gfCNCPoint4[1229] = {X 18.0872, Y 34.0798, Z -5.5000, A 0.000, B 0.000, C 0.000 }
gfCNCPoint4[1230] = {X 16.0874, Y 34.3007, Z -5.5000, A 0.000, B 0.000, C 0.000 }
gfCNCPoint4[1231] = {X 15.3633, Y 34.3534, Z -5.5000, A 0.000, B 0.000, C 0.000 }
gfCNCPoint4[1232] = {X 14.6390, Y 34.4040, Z -5.5000, A 0.000, B 0.000, C 0.000 }
gfCNCPoint4[1233] = {X 10.6873, Y 35.0236, Z -5.5000, A 0.000, B 0.000, C 0.000 }
gfCNCPoint4[1234] = {X 14.7700, Y 36.3195, Z -5.5000, A 0.000, B 0.000, C 0.000 }
gfCNCPoint4[1235] = {X 14.6336, Y 34.3242, Z -5.5000, A 0.000, B 0.000, C 0.000 }
gfCNCPoint4[1236] = {X 12.2421, Y 34.4763, Z -5.5000, A 0.000, B 0.000, C 0.000 }
gfCNCPoint4[1237] = {X 9.8492, Y 34.6056, Z -5.5000, A 0.000, B 0.000, C 0.000 }
gfCNCPoint4[1238] = {X 8.5938, Y 34.7145, Z -5.5000, A 0.000, B 0.000, C 0.000 }
gfCNCPoint4[1239] = {X 7.3613, Y 34.9767, Z -5.5000, A 0.000, B 0.000, C 0.000 }
gfCNCPoint4[1240] = {X 7.2805, Y 35.1981, Z -5.5000, A 0.000, B 0.000, C 0.000 }
gfCNCPoint4[1241] = {X 7.2526, Y 35.4321, Z -5.5000, A 0.000, B 0.000, C 0.000 }
gfCNCPoint4[1242] = {X 7.3219, Y 35.9823, Z -5.5000, A 0.000, B 0.000, C 0.000 }
gfCNCPoint4[1243] = {X 7.5291, Y 36.4967, Z -5.5000, A 0.000, B 0.000, C 0.000 }
gfCNCPoint4[1244] = {X 7.8606, Y 36.9413, Z -5.5000, A 0.000, B 0.000, C 0.000 }
gfCNCPoint4[1245] = {X 8.2944, Y 37.2868, Z -5.5000, A 0.000, B 0.000, C 0.000 }
gfCNCPoint4[1246] = {X 9.1221, Y 37.7063, Z -5.5000, A 0.000, B 0.000, C 0.000 }
gfCNCPoint4[1247] = {X 10.0031, Y 37.9977, Z -5.5000, A 0.000, B 0.000, C 0.000 }
gfCNCPoint4[1248] = {X 11.3365, Y 38.2429, Z -5.5000, A 0.000, B 0.000, C 0.000 }
gfCNCPoint4[1249] = {X 12.6902, Y 38.3190, Z -5.5000, A 0.000, B 0.000, C 0.000 }
gfCNCPoint4[1250] = {X 14.0427, Y 38.2248, Z -5.5000, A 0.000, B 0.000, C 0.000 }
gfCNCPoint4[1251] = {X 15.3727, Y 37.9617, Z -5.5000, A 0.000, B 0.000, C 0.000 }
gfCNCPoint4[1252] = {X 16.6593, Y 37.5340, Z -5.5000, A 0.000, B 0.000, C 0.000 }
gfCNCPoint4[1253] = {X 18.0880, Y 36.8591, Z -5.5000, A 0.000, B 0.000, C 0.000 }
gfCNCPoint4[1254] = {X 19.4300, Y 36.0248, Z -5.5000, A 0.000, B 0.000, C 0.000 }
gfCNCPoint4[1255] = {X 19.5226, Y 35.1553, Z -5.5000, A 0.000, B 0.000, C 0.000 }
gfCNCPoint4[1256] = {X 19.8019, Y 34.3266, Z -5.5000, A 0.000, B 0.000, C 0.000 }
gfCNCPoint4[1257] = {X 20.2547, Y 33.5784, Z -5.5000, A 0.000, B 0.000, C 0.000 }
gfCNCPoint4[1258] = {X 18.1812, Y 33.9846, Z -5.5000, A 0.000, B 0.000, C 0.000 }
gfCNCPoint4[1259] = {X 16.0816, Y 34.2210, Z -5.5000, A 0.000, B 0.000, C 0.000 }
gfCNCPoint4[1260] = {X 15.3577, Y 34.2736, Z -5.5000, A 0.000, B 0.000, C 0.000 }
gfCNCPoint4[1261] = {X 14.6336, Y 34.3242, Z -5.5000, A 0.000, B 0.000, C 0.000 }
gfCNCPoint4[1262] = {X 14.7700, Y 36.3195, Z -5.5000, A 0.000, B 0.000, C 0.000 }
gfCNCPoint4[1263] = {X 14.7700, Y 36.3195, Z -2.5000, A 0.000, B 0.000, C 0.000 }
gfCNCPoint4[1264] = {X 14.7700, Y 36.3195, Z 11.0000, A 0.000, B 0.000, C 0.000 }
gfCNCPoint4[1265] = {X 165.6772, Y 73.8165, Z 11.0000, A 0.000, B 0.000, C 0.000 }
gfCNCPoint4[1266] = {X 165.6772, Y 73.8165, Z -1.6667, A 0.000, B 0.000, C 0.000 }
gfCNCPoint4[1267] = {X 161.3996, Y 78.5670, Z -3.3796, A 0.000, B 0.000, C 0.000 }
gfCNCPoint4[1268] = {X 169.3132, Y 78.5670, Z -5.5000, A 0.000, B 0.000, C 0.000 }
gfCNCPoint4[1269] = {X 169.3132, Y 76.1670, Z -5.5000, A 0.000, B 0.000, C 0.000 }
gfCNCPoint4[1270] = {X 171.8361, Y 76.1670, Z -5.5000, A 0.000, B 0.000, C 0.000 }
gfCNCPoint4[1271] = {X 169.3147, Y 73.3634, Z -5.5000, A 0.000, B 0.000, C 0.000 }
gfCNCPoint4[1272] = {X 166.7903, Y 76.1670, Z -5.5000, A 0.000, B 0.000, C 0.000 }
gfCNCPoint4[1273] = {X 169.3132, Y 76.1670, Z -5.5000, A 0.000, B 0.000, C 0.000 }
gfCNCPoint4[1274] = {X 169.3132, Y 78.5670, Z -5.5000, A 0.000, B 0.000, C 0.000 }
gfCNCPoint4[1275] = {X 177.2224, Y 78.5670, Z -5.5000, A 0.000, B 0.000, C 0.000 }
gfCNCPoint4[1276] = {X 169.3158, Y 69.7756, Z -5.5000, A 0.000, B 0.000, C 0.000 }
gfCNCPoint4[1277] = {X 161.3996, Y 78.5670, Z -5.5000, A 0.000, B 0.000, C 0.000 }
gfCNCPoint4[1278] = {X 169.3132, Y 78.5670, Z -5.5000, A 0.000, B 0.000, C 0.000 }
gfCNCPoint4[1279] = {X 169.3132, Y 74.6470, Z -5.5000, A 0.000, B 0.000, C 0.000 }
gfCNCPoint4[1280] = {X 169.3132, Y 78.6470, Z -5.5000, A 0.000, B 0.000, C 0.000 }
gfCNCPoint4[1281] = {X 177.4019, Y 78.6470, Z -5.5000, A 0.000, B 0.000, C 0.000 }
gfCNCPoint4[1282] = {X 169.3159, Y 69.6560, Z -5.5000, A 0.000, B 0.000, C 0.000 }
gfCNCPoint4[1283] = {X 161.2199, Y 78.6470, Z -5.5000, A 0.000, B 0.000, C 0.000 }
gfCNCPoint4[1284] = {X 169.3132, Y 78.6470, Z -5.5000, A 0.000, B 0.000, C 0.000 }
gfCNCPoint4[1285] = {X 169.3132, Y 74.6470, Z -5.5000, A 0.000, B 0.000, C 0.000 }
gfCNCPoint4[1286] = {X 169.3132, Y 74.7270, Z -5.5000, A 0.000, B 0.000, C 0.000 }
gfCNCPoint4[1287] = {X 169.3132, Y 78.7270, Z -5.5000, A 0.000, B 0.000, C 0.000 }
gfCNCPoint4[1288] = {X 177.5814, Y 78.7270, Z -5.5000, A 0.000, B 0.000, C 0.000 }
gfCNCPoint4[1289] = {X 169.3159, Y 69.5364, Z -5.5000, A 0.000, B 0.000, C 0.000 }
gfCNCPoint4[1290] = {X 161.0403, Y 78.7270, Z -5.5000, A 0.000, B 0.000, C 0.000 }
gfCNCPoint4[1291] = {X 169.3132, Y 78.7270, Z -5.5000, A 0.000, B 0.000, C 0.000 }
gfCNCPoint4[1292] = {X 169.3132, Y 74.7270, Z -5.5000, A 0.000, B 0.000, C 0.000 }
gfCNCPoint4[1293] = {X 169.3132, Y 74.8070, Z -5.5000, A 0.000, B 0.000, C 0.000 }
gfCNCPoint4[1294] = {X 169.3132, Y 78.8070, Z -5.5000, A 0.000, B 0.000, C 0.000 }
gfCNCPoint4[1295] = {X 177.7610, Y 78.8070, Z -5.5000, A 0.000, B 0.000, C 0.000 }
gfCNCPoint4[1296] = {X 169.3159, Y 69.4168, Z -5.5000, A 0.000, B 0.000, C 0.000 }
gfCNCPoint4[1297] = {X 160.8606, Y 78.8070, Z -5.5000, A 0.000, B 0.000, C 0.000 }
gfCNCPoint4[1298] = {X 169.3132, Y 78.8070, Z -5.5000, A 0.000, B 0.000, C 0.000 }
gfCNCPoint4[1299] = {X 169.3132, Y 74.8070, Z -5.5000, A 0.000, B 0.000, C 0.000 }
gfCNCPoint4[1300] = {X 169.3132, Y 74.8870, Z -5.5000, A 0.000, B 0.000, C 0.000 }
gfCNCPoint4[1301] = {X 169.3132, Y 78.8870, Z -5.5000, A 0.000, B 0.000, C 0.000 }
gfCNCPoint4[1302] = {X 177.9405, Y 78.8870, Z -5.5000, A 0.000, B 0.000, C 0.000 }
gfCNCPoint4[1303] = {X 169.3160, Y 69.2972, Z -5.5000, A 0.000, B 0.000, C 0.000 }
gfCNCPoint4[1304] = {X 160.6809, Y 78.8870, Z -5.5000, A 0.000, B 0.000, C 0.000 }
gfCNCPoint4[1305] = {X 169.3132, Y 78.8870, Z -5.5000, A 0.000, B 0.000, C 0.000 }
gfCNCPoint4[1306] = {X 169.3132, Y 74.8870, Z -5.5000, A 0.000, B 0.000, C 0.000 }
gfCNCPoint4[1307] = {X 169.3132, Y 74.9670, Z -5.5000, A 0.000, B 0.000, C 0.000 }
gfCNCPoint4[1308] = {X 169.3132, Y 78.9670, Z -5.5000, A 0.000, B 0.000, C 0.000 }
gfCNCPoint4[1309] = {X 178.1201, Y 78.9670, Z -5.5000, A 0.000, B 0.000, C 0.000 }
gfCNCPoint4[1310] = {X 169.3160, Y 69.1776, Z -5.5000, A 0.000, B 0.000, C 0.000 }
gfCNCPoint4[1311] = {X 160.5012, Y 78.9670, Z -5.5000, A 0.000, B 0.000, C 0.000 }
gfCNCPoint4[1312] = {X 169.3132, Y 78.9670, Z -5.5000, A 0.000, B 0.000, C 0.000 }
gfCNCPoint4[1313] = {X 169.3132, Y 74.9670, Z -5.5000, A 0.000, B 0.000, C 0.000 }
gfCNCPoint4[1314] = {X 169.3132, Y 74.9670, Z -2.5000, A 0.000, B 0.000, C 0.000 }
gfCNCPoint4[1315] = {X 169.3132, Y 74.9670, Z 11.0000, A 0.000, B 0.000, C 0.000 }
gfCNCPoint4[1316] = {X 186.2281, Y 37.9121, Z 11.0000, A 0.000, B 0.000, C 0.000 }
gfCNCPoint4[1317] = {X 186.2281, Y 37.9121, Z -1.6667, A 0.000, B 0.000, C 0.000 }
gfCNCPoint4[1318] = {X 187.5897, Y 37.8323, Z -2.0321, A 0.000, B 0.000, C 0.000 }
gfCNCPoint4[1319] = {X 189.4169, Y 37.3859, Z -2.5361, A 0.000, B 0.000, C 0.000 }
gfCNCPoint4[1320] = {X 190.1421, Y 37.0740, Z -2.7476, A 0.000, B 0.000, C 0.000 }
gfCNCPoint4[1321] = {X 190.9803, Y 36.7135, Z -2.9922, A 0.000, B 0.000, C 0.000 }
gfCNCPoint4[1322] = {X 191.6914, Y 36.3240, Z -3.2094, A 0.000, B 0.000, C 0.000 }
gfCNCPoint4[1323] = {X 192.4466, Y 35.8118, Z -3.4539, A 0.000, B 0.000, C 0.000 }
gfCNCPoint4[1324] = {X 192.4699, Y 35.2976, Z -3.5918, A 0.000, B 0.000, C 0.000 }
gfCNCPoint4[1325] = {X 192.6312, Y 34.6351, Z -3.7745, A 0.000, B 0.000, C 0.000 }
gfCNCPoint4[1326] = {X 192.8468, Y 34.1677, Z -3.9124, A 0.000, B 0.000, C 0.000 }
gfCNCPoint4[1327] = {X 192.7389, Y 34.1929, Z -3.9421, A 0.000, B 0.000, C 0.000 }
gfCNCPoint4[1328] = {X 191.4080, Y 34.4432, Z -4.3050, A 0.000, B 0.000, C 0.000 }
gfCNCPoint4[1329] = {X 190.5815, Y 34.5495, Z -4.5283, A 0.000, B 0.000, C 0.000 }
gfCNCPoint4[1330] = {X 189.2271, Y 34.6445, Z -4.8921, A 0.000, B 0.000, C 0.000 }
gfCNCPoint4[1331] = {X 186.9627, Y 34.7836, Z -5.5000, A 0.000, B 0.000, C 0.000 }
gfCNCPoint4[1332] = {X 182.5757, Y 35.0529, Z -5.5000, A 0.000, B 0.000, C 0.000 }
gfCNCPoint4[1333] = {X 181.8176, Y 35.1403, Z -5.5000, A 0.000, B 0.000, C 0.000 }
gfCNCPoint4[1334] = {X 181.0731, Y 35.3082, Z -5.5000, A 0.000, B 0.000, C 0.000 }
gfCNCPoint4[1335] = {X 181.0650, Y 35.3823, Z -5.5000, A 0.000, B 0.000, C 0.000 }
gfCNCPoint4[1336] = {X 181.0651, Y 35.4570, Z -5.5000, A 0.000, B 0.000, C 0.000 }
gfCNCPoint4[1337] = {X 181.1578, Y 35.9998, Z -5.5000, A 0.000, B 0.000, C 0.000 }
gfCNCPoint4[1338] = {X 181.4149, Y 36.4869, Z -5.5000, A 0.000, B 0.000, C 0.000 }
gfCNCPoint4[1339] = {X 181.8107, Y 36.8698, Z -5.5000, A 0.000, B 0.000, C 0.000 }
gfCNCPoint4[1340] = {X 182.4284, Y 37.2226, Z -5.5000, A 0.000, B 0.000, C 0.000 }
gfCNCPoint4[1341] = {X 183.0886, Y 37.4872, Z -5.5000, A 0.000, B 0.000, C 0.000 }
gfCNCPoint4[1342] = {X 184.4948, Y 37.8011, Z -5.5000, A 0.000, B 0.000, C 0.000 }
gfCNCPoint4[1343] = {X 185.9310, Y 37.9170, Z -5.5000, A 0.000, B 0.000, C 0.000 }
gfCNCPoint4[1344] = {X 187.3693, Y 37.8327, Z -5.5000, A 0.000, B 0.000, C 0.000 }
gfCNCPoint4[1345] = {X 188.7821, Y 37.5499, Z -5.5000, A 0.000, B 0.000, C 0.000 }
gfCNCPoint4[1346] = {X 190.1421, Y 37.0740, Z -5.5000, A 0.000, B 0.000, C 0.000 }
gfCNCPoint4[1347] = {X 191.3243, Y 36.4976, Z -5.5000, A 0.000, B 0.000, C 0.000 }
gfCNCPoint4[1348] = {X 192.4466, Y 35.8118, Z -5.5000, A 0.000, B 0.000, C 0.000 }
gfCNCPoint4[1349] = {X 192.5670, Y 34.9703, Z -5.5000, A 0.000, B 0.000, C 0.000 }
gfCNCPoint4[1350] = {X 192.8468, Y 34.1677, Z -5.5000, A 0.000, B 0.000, C 0.000 }
gfCNCPoint4[1351] = {X 192.7389, Y 34.1929, Z -5.5000, A 0.000, B 0.000, C 0.000 }
gfCNCPoint4[1352] = {X 190.9895, Y 34.4696, Z -5.5000, A 0.000, B 0.000, C 0.000 }
gfCNCPoint4[1353] = {X 189.2271, Y 34.6445, Z -5.5000, A 0.000, B 0.000, C 0.000 }
gfCNCPoint4[1354] = {X 186.9627, Y 34.7836, Z -5.5000, A 0.000, B 0.000, C 0.000 }
gfCNCPoint4[1355] = {X 190.9564, Y 34.8075, Z -5.5000, A 0.000, B 0.000, C 0.000 }
gfCNCPoint4[1356] = {X 186.9578, Y 34.7037, Z -5.5000, A 0.000, B 0.000, C 0.000 }
gfCNCPoint4[1357] = {X 182.5708, Y 34.9731, Z -5.5000, A 0.000, B 0.000, C 0.000 }
gfCNCPoint4[1358] = {X 181.7800, Y 35.0656, Z -5.5000, A 0.000, B 0.000, C 0.000 }
gfCNCPoint4[1359] = {X 181.0042, Y 35.2447, Z -5.5000, A 0.000, B 0.000, C 0.000 }
gfCNCPoint4[1360] = {X 180.9874, Y 35.3482, Z -5.5000, A 0.000, B 0.000, C 0.000 }
gfCNCPoint4[1361] = {X 180.9850, Y 35.4530, Z -5.5000, A 0.000, B 0.000, C 0.000 }
gfCNCPoint4[1362] = {X 181.0811, Y 36.0228, Z -5.5000, A 0.000, B 0.000, C 0.000 }
gfCNCPoint4[1363] = {X 181.3503, Y 36.5341, Z -5.5000, A 0.000, B 0.000, C 0.000 }
gfCNCPoint4[1364] = {X 181.7656, Y 36.9358, Z -5.5000, A 0.000, B 0.000, C 0.000 }
gfCNCPoint4[1365] = {X 182.3936, Y 37.2947, Z -5.5000, A 0.000, B 0.000, C 0.000 }
gfCNCPoint4[1366] = {X 183.0649, Y 37.5636, Z -5.5000, A 0.000, B 0.000, C 0.000 }
gfCNCPoint4[1367] = {X 184.4822, Y 37.8801, Z -5.5000, A 0.000, B 0.000, C 0.000 }
gfCNCPoint4[1368] = {X 185.9296, Y 37.9970, Z -5.5000, A 0.000, B 0.000, C 0.000 }
gfCNCPoint4[1369] = {X 187.3792, Y 37.9121, Z -5.5000, A 0.000, B 0.000, C 0.000 }
gfCNCPoint4[1370] = {X 188.8031, Y 37.6271, Z -5.5000, A 0.000, B 0.000, C 0.000 }
gfCNCPoint4[1371] = {X 190.1737, Y 37.1475, Z -5.5000, A 0.000, B 0.000, C 0.000 }
gfCNCPoint4[1372] = {X 191.3805, Y 36.5581, Z -5.5000, A 0.000, B 0.000, C 0.000 }
gfCNCPoint4[1373] = {X 192.5249, Y 35.8553, Z -5.5000, A 0.000, B 0.000, C 0.000 }
gfCNCPoint4[1374] = {X 192.6602, Y 34.9276, Z -5.5000, A 0.000, B 0.000, C 0.000 }
gfCNCPoint4[1375] = {X 192.9924, Y 34.0510, Z -5.5000, A 0.000, B 0.000, C 0.000 }
gfCNCPoint4[1376] = {X 192.7315, Y 34.1128, Z -5.5000, A 0.000, B 0.000, C 0.000 }
gfCNCPoint4[1377] = {X 190.9841, Y 34.3897, Z -5.5000, A 0.000, B 0.000, C 0.000 }
gfCNCPoint4[1378] = {X 189.2236, Y 34.5646, Z -5.5000, A 0.000, B 0.000, C 0.000 }
gfCNCPoint4[1379] = {X 186.9578, Y 34.7037, Z -5.5000, A 0.000, B 0.000, C 0.000 }
gfCNCPoint4[1380] = {X 183.0018, Y 35.2959, Z -5.5000, A 0.000, B 0.000, C 0.000 }
gfCNCPoint4[1381] = {X 190.9515, Y 34.7276, Z -5.5000, A 0.000, B 0.000, C 0.000 }
gfCNCPoint4[1382] = {X 186.9529, Y 34.6239, Z -5.5000, A 0.000, B 0.000, C 0.000 }
gfCNCPoint4[1383] = {X 182.5658, Y 34.8932, Z -5.5000, A 0.000, B 0.000, C 0.000 }
gfCNCPoint4[1384] = {X 181.7439, Y 34.9907, Z -5.5000, A 0.000, B 0.000, C 0.000 }
gfCNCPoint4[1385] = {X 180.9383, Y 35.1806, Z -5.5000, A 0.000, B 0.000, C 0.000 }
gfCNCPoint4[1386] = {X 180.9104, Y 35.3165, Z -5.5000, A 0.000, B 0.000, C 0.000 }
gfCNCPoint4[1387] = {X 180.9051, Y 35.4551, Z -5.5000, A 0.000, B 0.000, C 0.000 }
gfCNCPoint4[1388] = {X 181.0057, Y 36.0496, Z -5.5000, A 0.000, B 0.000, C 0.000 }
gfCNCPoint4[1389] = {X 181.2869, Y 36.5829, Z -5.5000, A 0.000, B 0.000, C 0.000 }
gfCNCPoint4[1390] = {X 181.7205, Y 37.0019, Z -5.5000, A 0.000, B 0.000, C 0.000 }
gfCNCPoint4[1391] = {X 182.3588, Y 37.3667, Z -5.5000, A 0.000, B 0.000, C 0.000 }
gfCNCPoint4[1392] = {X 183.0413, Y 37.6400, Z -5.5000, A 0.000, B 0.000, C 0.000 }
gfCNCPoint4[1393] = {X 184.4695, Y 37.9591, Z -5.5000, A 0.000, B 0.000, C 0.000 }
gfCNCPoint4[1394] = {X 185.9281, Y 38.0770, Z -5.5000, A 0.000, B 0.000, C 0.000 }
gfCNCPoint4[1395] = {X 187.3890, Y 37.9915, Z -5.5000, A 0.000, B 0.000, C 0.000 }
gfCNCPoint4[1396] = {X 188.8240, Y 37.7043, Z -5.5000, A 0.000, B 0.000, C 0.000 }
gfCNCPoint4[1397] = {X 190.2053, Y 37.2210, Z -5.5000, A 0.000, B 0.000, C 0.000 }
gfCNCPoint4[1398] = {X 191.4368, Y 36.6184, Z -5.5000, A 0.000, B 0.000, C 0.000 }
gfCNCPoint4[1399] = {X 192.6036, Y 35.8984, Z -5.5000, A 0.000, B 0.000, C 0.000 }
gfCNCPoint4[1400] = {X 192.6773, Y 35.2164, Z -5.5000, A 0.000, B 0.000, C 0.000 }
gfCNCPoint4[1401] = {X 192.8599, Y 34.5552, Z -5.5000, A 0.000, B 0.000, C 0.000 }
gfCNCPoint4[1402] = {X 193.1467, Y 33.9322, Z -5.5000, A 0.000, B 0.000, C 0.000 }
gfCNCPoint4[1403] = {X 192.7149, Y 34.0346, Z -5.5000, A 0.000, B 0.000, C 0.000 }
gfCNCPoint4[1404] = {X 190.9731, Y 34.3104, Z -5.5000, A 0.000, B 0.000, C 0.000 }
gfCNCPoint4[1405] = {X 189.2183, Y 34.4848, Z -5.5000, A 0.000, B 0.000, C 0.000 }
gfCNCPoint4[1406] = {X 186.9529, Y 34.6239, Z -5.5000, A 0.000, B 0.000, C 0.000 }
gfCNCPoint4[1407] = {X 182.9969, Y 35.2160, Z -5.5000, A 0.000, B 0.000, C 0.000 }
gfCNCPoint4[1408] = {X 190.9466, Y 34.6478, Z -5.5000, A 0.000, B 0.000, C 0.000 }
gfCNCPoint4[1409] = {X 186.9480, Y 34.5440, Z -5.5000, A 0.000, B 0.000, C 0.000 }
gfCNCPoint4[1410] = {X 182.5609, Y 34.8134, Z -5.5000, A 0.000, B 0.000, C 0.000 }
gfCNCPoint4[1411] = {X 181.7092, Y 34.9156, Z -5.5000, A 0.000, B 0.000, C 0.000 }
gfCNCPoint4[1412] = {X 180.8750, Y 35.1161, Z -5.5000, A 0.000, B 0.000, C 0.000 }
gfCNCPoint4[1413] = {X 180.8340, Y 35.2843, Z -5.5000, A 0.000, B 0.000, C 0.000 }
gfCNCPoint4[1414] = {X 180.8251, Y 35.4572, Z -5.5000, A 0.000, B 0.000, C 0.000 }
gfCNCPoint4[1415] = {X 180.9303, Y 36.0764, Z -5.5000, A 0.000, B 0.000, C 0.000 }
gfCNCPoint4[1416] = {X 181.2235, Y 36.6318, Z -5.5000, A 0.000, B 0.000, C 0.000 }
gfCNCPoint4[1417] = {X 181.6754, Y 37.0680, Z -5.5000, A 0.000, B 0.000, C 0.000 }
gfCNCPoint4[1418] = {X 182.3240, Y 37.4387, Z -5.5000, A 0.000, B 0.000, C 0.000 }
gfCNCPoint4[1419] = {X 183.0176, Y 37.7165, Z -5.5000, A 0.000, B 0.000, C 0.000 }
gfCNCPoint4[1420] = {X 184.4568, Y 38.0381, Z -5.5000, A 0.000, B 0.000, C 0.000 }
gfCNCPoint4[1421] = {X 185.9267, Y 38.1570, Z -5.5000, A 0.000, B 0.000, C 0.000 }
gfCNCPoint4[1422] = {X 187.3989, Y 38.0709, Z -5.5000, A 0.000, B 0.000, C 0.000 }
gfCNCPoint4[1423] = {X 188.8449, Y 37.7815, Z -5.5000, A 0.000, B 0.000, C 0.000 }
gfCNCPoint4[1424] = {X 190.2369, Y 37.2945, Z -5.5000, A 0.000, B 0.000, C 0.000 }
gfCNCPoint4[1425] = {X 191.4934, Y 36.6785, Z -5.5000, A 0.000, B 0.000, C 0.000 }
gfCNCPoint4[1426] = {X 192.6827, Y 35.9410, Z -5.5000, A 0.000, B 0.000, C 0.000 }
gfCNCPoint4[1427] = {X 192.7626, Y 35.1969, Z -5.5000, A 0.000, B 0.000, C 0.000 }
gfCNCPoint4[1428] = {X 192.9745, Y 34.4791, Z -5.5000, A 0.000, B 0.000, C 0.000 }
gfCNCPoint4[1429] = {X 193.3115, Y 33.8109, Z -5.5000, A 0.000, B 0.000, C 0.000 }
gfCNCPoint4[1430] = {X 192.6982, Y 33.9563, Z -5.5000, A 0.000, B 0.000, C 0.000 }
gfCNCPoint4[1431] = {X 190.9622, Y 34.2312, Z -5.5000, A 0.000, B 0.000, C 0.000 }
gfCNCPoint4[1432] = {X 189.2131, Y 34.4049, Z -5.5000, A 0.000, B 0.000, C 0.000 }
gfCNCPoint4[1433] = {X 186.9480, Y 34.5440, Z -5.5000, A 0.000, B 0.000, C 0.000 }
gfCNCPoint4[1434] = {X 182.9920, Y 35.1362, Z -5.5000, A 0.000, B 0.000, C 0.000 }
gfCNCPoint4[1435] = {X 190.9417, Y 34.5679, Z -5.5000, A 0.000, B 0.000, C 0.000 }
gfCNCPoint4[1436] = {X 186.9431, Y 34.4642, Z -5.5000, A 0.000, B 0.000, C 0.000 }
gfCNCPoint4[1437] = {X 182.5560, Y 34.7335, Z -5.5000, A 0.000, B 0.000, C 0.000 }
gfCNCPoint4[1438] = {X 181.6754, Y 34.8405, Z -5.5000, A 0.000, B 0.000, C 0.000 }
gfCNCPoint4[1439] = {X 180.8137, Y 35.0511, Z -5.5000, A 0.000, B 0.000, C 0.000 }
gfCNCPoint4[1440] = {X 180.7581, Y 35.2516, Z -5.5000, A 0.000, B 0.000, C 0.000 }
gfCNCPoint4[1441] = {X 180.7451, Y 35.4593, Z -5.5000, A 0.000, B 0.000, C 0.000 }
gfCNCPoint4[1442] = {X 180.8550, Y 36.1032, Z -5.5000, A 0.000, B 0.000, C 0.000 }
gfCNCPoint4[1443] = {X 181.1602, Y 36.6806, Z -5.5000, A 0.000, B 0.000, C 0.000 }
gfCNCPoint4[1444] = {X 181.6303, Y 37.1341, Z -5.5000, A 0.000, B 0.000, C 0.000 }
gfCNCPoint4[1445] = {X 182.2892, Y 37.5108, Z -5.5000, A 0.000, B 0.000, C 0.000 }
gfCNCPoint4[1446] = {X 182.9939, Y 37.7929, Z -5.5000, A 0.000, B 0.000, C 0.000 }
gfCNCPoint4[1447] = {X 184.4441, Y 38.1170, Z -5.5000, A 0.000, B 0.000, C 0.000 }
gfCNCPoint4[1448] = {X 185.9253, Y 38.2370, Z -5.5000, A 0.000, B 0.000, C 0.000 }
gfCNCPoint4[1449] = {X 187.4087, Y 38.1503, Z -5.5000, A 0.000, B 0.000, C 0.000 }
gfCNCPoint4[1450] = {X 188.8659, Y 37.8588, Z -5.5000, A 0.000, B 0.000, C 0.000 }
gfCNCPoint4[1451] = {X 190.2685, Y 37.3680, Z -5.5000, A 0.000, B 0.000, C 0.000 }
gfCNCPoint4[1452] = {X 191.5503, Y 36.7385, Z -5.5000, A 0.000, B 0.000, C 0.000 }
gfCNCPoint4[1453] = {X 192.7622, Y 35.9832, Z -5.5000, A 0.000, B 0.000, C 0.000 }
gfCNCPoint4[1454] = {X 192.8358, Y 35.2393, Z -5.5000, A 0.000, B 0.000, C 0.000 }
gfCNCPoint4[1455] = {X 193.0438, Y 34.5212, Z -5.5000, A 0.000, B 0.000, C 0.000 }
gfCNCPoint4[1456] = {X 193.3794, Y 33.8532, Z -5.5000, A 0.000, B 0.000, C 0.000 }
gfCNCPoint4[1457] = {X 193.4225, Y 33.7856, Z -5.5000, A 0.000, B 0.000, C 0.000 }
gfCNCPoint4[1458] = {X 193.4669, Y 33.7188, Z -5.5000, A 0.000, B 0.000, C 0.000 }
gfCNCPoint4[1459] = {X 193.3657, Y 33.7158, Z -5.5000, A 0.000, B 0.000, C 0.000 }
gfCNCPoint4[1460] = {X 192.6816, Y 33.8780, Z -5.5000, A 0.000, B 0.000, C 0.000 }
gfCNCPoint4[1461] = {X 190.9512, Y 34.1519, Z -5.5000, A 0.000, B 0.000, C 0.000 }
gfCNCPoint4[1462] = {X 189.2078, Y 34.3251, Z -5.5000, A 0.000, B 0.000, C 0.000 }
gfCNCPoint4[1463] = {X 186.9431, Y 34.4642, Z -5.5000, A 0.000, B 0.000, C 0.000 }
gfCNCPoint4[1464] = {X 182.9871, Y 35.0564, Z -5.5000, A 0.000, B 0.000, C 0.000 }
gfCNCPoint4[1465] = {X 190.9306, Y 34.1392, Z -5.5000, A 0.000, B 0.000, C 0.000 }
gfCNCPoint4[1466] = {X 186.9382, Y 34.3843, Z -5.5000, A 0.000, B 0.000, C 0.000 }
gfCNCPoint4[1467] = {X 182.5511, Y 34.6537, Z -5.5000, A 0.000, B 0.000, C 0.000 }
gfCNCPoint4[1468] = {X 181.6425, Y 34.7652, Z -5.5000, A 0.000, B 0.000, C 0.000 }
gfCNCPoint4[1469] = {X 180.7541, Y 34.9859, Z -5.5000, A 0.000, B 0.000, C 0.000 }
gfCNCPoint4[1470] = {X 180.6827, Y 35.2186, Z -5.5000, A 0.000, B 0.000, C 0.000 }
gfCNCPoint4[1471] = {X 180.6651, Y 35.4613, Z -5.5000, A 0.000, B 0.000, C 0.000 }
gfCNCPoint4[1472] = {X 180.7796, Y 36.1299, Z -5.5000, A 0.000, B 0.000, C 0.000 }
gfCNCPoint4[1473] = {X 181.0968, Y 36.7295, Z -5.5000, A 0.000, B 0.000, C 0.000 }
gfCNCPoint4[1474] = {X 181.5852, Y 37.2002, Z -5.5000, A 0.000, B 0.000, C 0.000 }
gfCNCPoint4[1475] = {X 182.2545, Y 37.5828, Z -5.5000, A 0.000, B 0.000, C 0.000 }
gfCNCPoint4[1476] = {X 182.9702, Y 37.8693, Z -5.5000, A 0.000, B 0.000, C 0.000 }
gfCNCPoint4[1477] = {X 184.4314, Y 38.1960, Z -5.5000, A 0.000, B 0.000, C 0.000 }
gfCNCPoint4[1478] = {X 185.9238, Y 38.3169, Z -5.5000, A 0.000, B 0.000, C 0.000 }
gfCNCPoint4[1479] = {X 187.4186, Y 38.2297, Z -5.5000, A 0.000, B 0.000, C 0.000 }
gfCNCPoint4[1480] = {X 188.8868, Y 37.9360, Z -5.5000, A 0.000, B 0.000, C 0.000 }
gfCNCPoint4[1481] = {X 190.3001, Y 37.4415, Z -5.5000, A 0.000, B 0.000, C 0.000 }
gfCNCPoint4[1482] = {X 191.6073, Y 36.7982, Z -5.5000, A 0.000, B 0.000, C 0.000 }
gfCNCPoint4[1483] = {X 192.8422, Y 36.0250, Z -5.5000, A 0.000, B 0.000, C 0.000 }
gfCNCPoint4[1484] = {X 192.9290, Y 35.1818, Z -5.5000, A 0.000, B 0.000, C 0.000 }
gfCNCPoint4[1485] = {X 193.1917, Y 34.3757, Z -5.5000, A 0.000, B 0.000, C 0.000 }
gfCNCPoint4[1486] = {X 193.6183, Y 33.6431, Z -5.5000, A 0.000, B 0.000, C 0.000 }
gfCNCPoint4[1487] = {X 193.3575, Y 33.6356, Z -5.5000, A 0.000, B 0.000, C 0.000 }
gfCNCPoint4[1488] = {X 192.6650, Y 33.7997, Z -5.5000, A 0.000, B 0.000, C 0.000 }
gfCNCPoint4[1489] = {X 190.9402, Y 34.0727, Z -5.5000, A 0.000, B 0.000, C 0.000 }
gfCNCPoint4[1490] = {X 189.2026, Y 34.2453, Z -5.5000, A 0.000, B 0.000, C 0.000 }
gfCNCPoint4[1491] = {X 186.9382, Y 34.3843, Z -5.5000, A 0.000, B 0.000, C 0.000 }
gfCNCPoint4[1492] = {X 182.9457, Y 34.6295, Z -5.5000, A 0.000, B 0.000, C 0.000 }
gfCNCPoint4[1493] = {X 182.9457, Y 34.6295, Z -2.5000, A 0.000, B 0.000, C 0.000 }
gfCNCPoint4[1494] = {X 182.9457, Y 34.6295, Z 11.0000, A 0.000, B 0.000, C 0.000 }
gfCNCPoint4[1495] = {X 188.4977, Y 19.4674, Z 11.0000, A 0.000, B 0.000, C 0.000 }
gfCNCPoint4[1496] = {X 188.4977, Y 19.4674, Z -1.6667, A 0.000, B 0.000, C 0.000 }
gfCNCPoint4[1497] = {X 188.3884, Y 19.4288, Z -1.6977, A 0.000, B 0.000, C 0.000 }
gfCNCPoint4[1498] = {X 187.7714, Y 19.3602, Z -1.8641, A 0.000, B 0.000, C 0.000 }
gfCNCPoint4[1499] = {X 186.9109, Y 19.2603, Z -2.0962, A 0.000, B 0.000, C 0.000 }
gfCNCPoint4[1500] = {X 184.5930, Y 19.3678, Z -2.7179, A 0.000, B 0.000, C 0.000 }
gfCNCPoint4[1501] = {X 183.7426, Y 19.5475, Z -2.9508, A 0.000, B 0.000, C 0.000 }
gfCNCPoint4[1502] = {X 183.0434, Y 19.6900, Z -3.1420, A 0.000, B 0.000, C 0.000 }
gfCNCPoint4[1503] = {X 182.0227, Y 20.0615, Z -3.4331, A 0.000, B 0.000, C 0.000 }
gfCNCPoint4[1504] = {X 181.3955, Y 20.4017, Z -3.6243, A 0.000, B 0.000, C 0.000 }
gfCNCPoint4[1505] = {X 181.3395, Y 20.9133, Z -3.7622, A 0.000, B 0.000, C 0.000 }
gfCNCPoint4[1506] = {X 180.8650, Y 22.1260, Z -4.1111, A 0.000, B 0.000, C 0.000 }
gfCNCPoint4[1507] = {X 180.5589, Y 22.5398, Z -4.2490, A 0.000, B 0.000, C 0.000 }
gfCNCPoint4[1508] = {X 182.2916, Y 22.3338, Z -4.7166, A 0.000, B 0.000, C 0.000 }
gfCNCPoint4[1509] = {X 182.5945, Y 22.3093, Z -4.7980, A 0.000, B 0.000, C 0.000 }
gfCNCPoint4[1510] = {X 184.3413, Y 22.2331, Z -5.2665, A 0.000, B 0.000, C 0.000 }
gfCNCPoint4[1511] = {X 184.7768, Y 22.2180, Z -5.3833, A 0.000, B 0.000, C 0.000 }
gfCNCPoint4[1512] = {X 185.2121, Y 22.1996, Z -5.5000, A 0.000, B 0.000, C 0.000 }
gfCNCPoint4[1513] = {X 187.5424, Y 22.0772, Z -5.5000, A 0.000, B 0.000, C 0.000 }
gfCNCPoint4[1514] = {X 189.8697, Y 21.9071, Z -5.5000, A 0.000, B 0.000, C 0.000 }
gfCNCPoint4[1515] = {X 190.4712, Y 21.8307, Z -5.5000, A 0.000, B 0.000, C 0.000 }
gfCNCPoint4[1516] = {X 191.0583, Y 21.6794, Z -5.5000, A 0.000, B 0.000, C 0.000 }
gfCNCPoint4[1517] = {X 191.0680, Y 21.1638, Z -5.5000, A 0.000, B 0.000, C 0.000 }
gfCNCPoint4[1518] = {X 190.8724, Y 20.6867, Z -5.5000, A 0.000, B 0.000, C 0.000 }
gfCNCPoint4[1519] = {X 190.5034, Y 20.3264, Z -5.5000, A 0.000, B 0.000, C 0.000 }
gfCNCPoint4[1520] = {X 189.6458, Y 19.8657, Z -5.5000, A 0.000, B 0.000, C 0.000 }
gfCNCPoint4[1521] = {X 188.7280, Y 19.5411, Z -5.5000, A 0.000, B 0.000, C 0.000 }
gfCNCPoint4[1522] = {X 187.7714, Y 19.3602, Z -5.5000, A 0.000, B 0.000, C 0.000 }
gfCNCPoint4[1523] = {X 186.4243, Y 19.2771, Z -5.5000, A 0.000, B 0.000, C 0.000 }
gfCNCPoint4[1524] = {X 185.0761, Y 19.3398, Z -5.5000, A 0.000, B 0.000, C 0.000 }
gfCNCPoint4[1525] = {X 183.7426, Y 19.5475, Z -5.5000, A 0.000, B 0.000, C 0.000 }
gfCNCPoint4[1526] = {X 182.5374, Y 19.8876, Z -5.5000, A 0.000, B 0.000, C 0.000 }
gfCNCPoint4[1527] = {X 181.3955, Y 20.4017, Z -5.5000, A 0.000, B 0.000, C 0.000 }
gfCNCPoint4[1528] = {X 181.2441, Y 21.1600, Z -5.5000, A 0.000, B 0.000, C 0.000 }
gfCNCPoint4[1529] = {X 180.9624, Y 21.8801, Z -5.5000, A 0.000, B 0.000, C 0.000 }
gfCNCPoint4[1530] = {X 180.5589, Y 22.5398, Z -5.5000, A 0.000, B 0.000, C 0.000 }
gfCNCPoint4[1531] = {X 182.4472, Y 22.3511, Z -5.5000, A 0.000, B 0.000, C 0.000 }
gfCNCPoint4[1532] = {X 184.3413, Y 22.2331, Z -5.5000, A 0.000, B 0.000, C 0.000 }
gfCNCPoint4[1533] = {X 184.7767, Y 22.2172, Z -5.5000, A 0.000, B 0.000, C 0.000 }
gfCNCPoint4[1534] = {X 185.2121, Y 22.1996, Z -5.5000, A 0.000, B 0.000, C 0.000 }
gfCNCPoint4[1535] = {X 181.2195, Y 22.0997, Z -5.5000, A 0.000, B 0.000, C 0.000 }
gfCNCPoint4[1536] = {X 185.2155, Y 22.2796, Z -5.5000, A 0.000, B 0.000, C 0.000 }
gfCNCPoint4[1537] = {X 187.5451, Y 22.1571, Z -5.5000, A 0.000, B 0.000, C 0.000 }
gfCNCPoint4[1538] = {X 189.8717, Y 21.9871, Z -5.5000, A 0.000, B 0.000, C 0.000 }
gfCNCPoint4[1539] = {X 190.5066, Y 21.9053, Z -5.5000, A 0.000, B 0.000, C 0.000 }
gfCNCPoint4[1540] = {X 191.1255, Y 21.7415, Z -5.5000, A 0.000, B 0.000, C 0.000 }
gfCNCPoint4[1541] = {X 191.1519, Y 21.1791, Z -5.5000, A 0.000, B 0.000, C 0.000 }
gfCNCPoint4[1542] = {X 190.9471, Y 20.6547, Z -5.5000, A 0.000, B 0.000, C 0.000 }
gfCNCPoint4[1543] = {X 190.5465, Y 20.2590, Z -5.5000, A 0.000, B 0.000, C 0.000 }
gfCNCPoint4[1544] = {X 189.6788, Y 19.7928, Z -5.5000, A 0.000, B 0.000, C 0.000 }
gfCNCPoint4[1545] = {X 188.7501, Y 19.4642, Z -5.5000, A 0.000, B 0.000, C 0.000 }
gfCNCPoint4[1546] = {X 187.7823, Y 19.2810, Z -5.5000, A 0.000, B 0.000, C 0.000 }
gfCNCPoint4[1547] = {X 186.4270, Y 19.1971, Z -5.5000, A 0.000, B 0.000, C 0.000 }
gfCNCPoint4[1548] = {X 185.0706, Y 19.2600, Z -5.5000, A 0.000, B 0.000, C 0.000 }
gfCNCPoint4[1549] = {X 183.7289, Y 19.4687, Z -5.5000, A 0.000, B 0.000, C 0.000 }
gfCNCPoint4[1550] = {X 182.4920, Y 19.8190, Z -5.5000, A 0.000, B 0.000, C 0.000 }
gfCNCPoint4[1551] = {X 181.3215, Y 20.3509, Z -5.5000, A 0.000, B 0.000, C 0.000 }
gfCNCPoint4[1552] = {X 181.1593, Y 21.1707, Z -5.5000, A 0.000, B 0.000, C 0.000 }
gfCNCPoint4[1553] = {X 180.8423, Y 21.9440, Z -5.5000, A 0.000, B 0.000, C 0.000 }
gfCNCPoint4[1554] = {X 180.3823, Y 22.6417, Z -5.5000, A 0.000, B 0.000, C 0.000 }
gfCNCPoint4[1555] = {X 182.3593, Y 22.4386, Z -5.5000, A 0.000, B 0.000, C 0.000 }
gfCNCPoint4[1556] = {X 184.3427, Y 22.3131, Z -5.5000, A 0.000, B 0.000, C 0.000 }
gfCNCPoint4[1557] = {X 184.7791, Y 22.2972, Z -5.5000, A 0.000, B 0.000, C 0.000 }
gfCNCPoint4[1558] = {X 185.2155, Y 22.2796, Z -5.5000, A 0.000, B 0.000, C 0.000 }
gfCNCPoint4[1559] = {X 189.1819, Y 21.7628, Z -5.5000, A 0.000, B 0.000, C 0.000 }
gfCNCPoint4[1560] = {X 181.2229, Y 22.1796, Z -5.5000, A 0.000, B 0.000, C 0.000 }
gfCNCPoint4[1561] = {X 185.2188, Y 22.3595, Z -5.5000, A 0.000, B 0.000, C 0.000 }
gfCNCPoint4[1562] = {X 187.5497, Y 22.2370, Z -5.5000, A 0.000, B 0.000, C 0.000 }
gfCNCPoint4[1563] = {X 189.8775, Y 22.0669, Z -5.5000, A 0.000, B 0.000, C 0.000 }
gfCNCPoint4[1564] = {X 190.5433, Y 21.9796, Z -5.5000, A 0.000, B 0.000, C 0.000 }
gfCNCPoint4[1565] = {X 191.1912, Y 21.8036, Z -5.5000, A 0.000, B 0.000, C 0.000 }
gfCNCPoint4[1566] = {X 191.2489, Y 21.3478, Z -5.5000, A 0.000, B 0.000, C 0.000 }
gfCNCPoint4[1567] = {X 191.1594, Y 20.8973, Z -5.5000, A 0.000, B 0.000, C 0.000 }
gfCNCPoint4[1568] = {X 190.9318, Y 20.4982, Z -5.5000, A 0.000, B 0.000, C 0.000 }
gfCNCPoint4[1569] = {X 190.5897, Y 20.1917, Z -5.5000, A 0.000, B 0.000, C 0.000 }
gfCNCPoint4[1570] = {X 189.7112, Y 19.7196, Z -5.5000, A 0.000, B 0.000, C 0.000 }
gfCNCPoint4[1571] = {X 188.7710, Y 19.3870, Z -5.5000, A 0.000, B 0.000, C 0.000 }
gfCNCPoint4[1572] = {X 187.7911, Y 19.2014, Z -5.5000, A 0.000, B 0.000, C 0.000 }
gfCNCPoint4[1573] = {X 186.4273, Y 19.1171, Z -5.5000, A 0.000, B 0.000, C 0.000 }
gfCNCPoint4[1574] = {X 185.0625, Y 19.1804, Z -5.5000, A 0.000, B 0.000, C 0.000 }
gfCNCPoint4[1575] = {X 183.7123, Y 19.3904, Z -5.5000, A 0.000, B 0.000, C 0.000 }
gfCNCPoint4[1576] = {X 182.4464, Y 19.7506, Z -5.5000, A 0.000, B 0.000, C 0.000 }
gfCNCPoint4[1577] = {X 181.2500, Y 20.2990, Z -5.5000, A 0.000, B 0.000, C 0.000 }
gfCNCPoint4[1578] = {X 181.2397, Y 20.3528, Z -5.5000, A 0.000, B 0.000, C 0.000 }
gfCNCPoint4[1579] = {X 181.0599, Y 21.2186, Z -5.5000, A 0.000, B 0.000, C 0.000 }
gfCNCPoint4[1580] = {X 180.7044, Y 22.0282, Z -5.5000, A 0.000, B 0.000, C 0.000 }
gfCNCPoint4[1581] = {X 180.1886, Y 22.7465, Z -5.5000, A 0.000, B 0.000, C 0.000 }
gfCNCPoint4[1582] = {X 182.2636, Y 22.5269, Z -5.5000, A 0.000, B 0.000, C 0.000 }
gfCNCPoint4[1583] = {X 184.3458, Y 22.3931, Z -5.5000, A 0.000, B 0.000, C 0.000 }
gfCNCPoint4[1584] = {X 184.7824, Y 22.3771, Z -5.5000, A 0.000, B 0.000, C 0.000 }
gfCNCPoint4[1585] = {X 185.2188, Y 22.3595, Z -5.5000, A 0.000, B 0.000, C 0.000 }
gfCNCPoint4[1586] = {X 189.1853, Y 21.8427, Z -5.5000, A 0.000, B 0.000, C 0.000 }
gfCNCPoint4[1587] = {X 181.2263, Y 22.2596, Z -5.5000, A 0.000, B 0.000, C 0.000 }
gfCNCPoint4[1588] = {X 185.2222, Y 22.4394, Z -5.5000, A 0.000, B 0.000, C 0.000 }
gfCNCPoint4[1589] = {X 187.5543, Y 22.3169, Z -5.5000, A 0.000, B 0.000, C 0.000 }
gfCNCPoint4[1590] = {X 189.8833, Y 22.1467, Z -5.5000, A 0.000, B 0.000, C 0.000 }
gfCNCPoint4[1591] = {X 190.5793, Y 22.0540, Z -5.5000, A 0.000, B 0.000, C 0.000 }
gfCNCPoint4[1592] = {X 191.2557, Y 21.8658, Z -5.5000, A 0.000, B 0.000, C 0.000 }
gfCNCPoint4[1593] = {X 191.3296, Y 21.3761, Z -5.5000, A 0.000, B 0.000, C 0.000 }
gfCNCPoint4[1594] = {X 191.2414, Y 20.8887, Z -5.5000, A 0.000, B 0.000, C 0.000 }
gfCNCPoint4[1595] = {X 191.0006, Y 20.4560, Z -5.5000, A 0.000, B 0.000, C 0.000 }
gfCNCPoint4[1596] = {X 190.6328, Y 20.1243, Z -5.5000, A 0.000, B 0.000, C 0.000 }
gfCNCPoint4[1597] = {X 189.7435, Y 19.6465, Z -5.5000, A 0.000, B 0.000, C 0.000 }
gfCNCPoint4[1598] = {X 188.7918, Y 19.3097, Z -5.5000, A 0.000, B 0.000, C 0.000 }
gfCNCPoint4[1599] = {X 187.7999, Y 19.1219, Z -5.5000, A 0.000, B 0.000, C 0.000 }
gfCNCPoint4[1600] = {X 186.4277, Y 19.0371, Z -5.5000, A 0.000, B 0.000, C 0.000 }
gfCNCPoint4[1601] = {X 185.0543, Y 19.1008, Z -5.5000, A 0.000, B 0.000, C 0.000 }
gfCNCPoint4[1602] = {X 183.6958, Y 19.3121, Z -5.5000, A 0.000, B 0.000, C 0.000 }
gfCNCPoint4[1603] = {X 182.4008, Y 19.6821, Z -5.5000, A 0.000, B 0.000, C 0.000 }
gfCNCPoint4[1604] = {X 181.1784, Y 20.2473, Z -5.5000, A 0.000, B 0.000, C 0.000 }
gfCNCPoint4[1605] = {X 181.1605, Y 20.3413, Z -5.5000, A 0.000, B 0.000, C 0.000 }
gfCNCPoint4[1606] = {X 180.9651, Y 21.2476, Z -5.5000, A 0.000, B 0.000, C 0.000 }
gfCNCPoint4[1607] = {X 180.5738, Y 22.0881, Z -5.5000, A 0.000, B 0.000, C 0.000 }
gfCNCPoint4[1608] = {X 180.0060, Y 22.8211, Z -5.5000, A 0.000, B 0.000, C 0.000 }
gfCNCPoint4[1609] = {X 180.1925, Y 22.8266, Z -5.5000, A 0.000, B 0.000, C 0.000 }
gfCNCPoint4[1610] = {X 182.2671, Y 22.6069, Z -5.5000, A 0.000, B 0.000, C 0.000 }
gfCNCPoint4[1611] = {X 184.3489, Y 22.4730, Z -5.5000, A 0.000, B 0.000, C 0.000 }
gfCNCPoint4[1612] = {X 184.7856, Y 22.4571, Z -5.5000, A 0.000, B 0.000, C 0.000 }
gfCNCPoint4[1613] = {X 185.2222, Y 22.4394, Z -5.5000, A 0.000, B 0.000, C 0.000 }
gfCNCPoint4[1614] = {X 189.1887, Y 21.9226, Z -5.5000, A 0.000, B 0.000, C 0.000 }
gfCNCPoint4[1615] = {X 181.2297, Y 22.3395, Z -5.5000, A 0.000, B 0.000, C 0.000 }
gfCNCPoint4[1616] = {X 185.2256, Y 22.5193, Z -5.5000, A 0.000, B 0.000, C 0.000 }
gfCNCPoint4[1617] = {X 187.5589, Y 22.3967, Z -5.5000, A 0.000, B 0.000, C 0.000 }
gfCNCPoint4[1618] = {X 189.8892, Y 22.2265, Z -5.5000, A 0.000, B 0.000, C 0.000 }
gfCNCPoint4[1619] = {X 190.6148, Y 22.1283, Z -5.5000, A 0.000, B 0.000, C 0.000 }
gfCNCPoint4[1620] = {X 191.3191, Y 21.9280, Z -5.5000, A 0.000, B 0.000, C 0.000 }
gfCNCPoint4[1621] = {X 191.4098, Y 21.4046, Z -5.5000, A 0.000, B 0.000, C 0.000 }
gfCNCPoint4[1622] = {X 191.3233, Y 20.8805, Z -5.5000, A 0.000, B 0.000, C 0.000 }
gfCNCPoint4[1623] = {X 191.0693, Y 20.4140, Z -5.5000, A 0.000, B 0.000, C 0.000 }
gfCNCPoint4[1624] = {X 190.6760, Y 20.0569, Z -5.5000, A 0.000, B 0.000, C 0.000 }
gfCNCPoint4[1625] = {X 189.7759, Y 19.5733, Z -5.5000, A 0.000, B 0.000, C 0.000 }
gfCNCPoint4[1626] = {X 188.8127, Y 19.2325, Z -5.5000, A 0.000, B 0.000, C 0.000 }
gfCNCPoint4[1627] = {X 187.8088, Y 19.0424, Z -5.5000, A 0.000, B 0.000, C 0.000 }
gfCNCPoint4[1628] = {X 186.4280, Y 18.9571, Z -5.5000, A 0.000, B 0.000, C 0.000 }
gfCNCPoint4[1629] = {X 185.0462, Y 19.0212, Z -5.5000, A 0.000, B 0.000, C 0.000 }
gfCNCPoint4[1630] = {X 183.6792, Y 19.2339, Z -5.5000, A 0.000, B 0.000, C 0.000 }
gfCNCPoint4[1631] = {X 182.3552, Y 19.6138, Z -5.5000, A 0.000, B 0.000, C 0.000 }
gfCNCPoint4[1632] = {X 181.1068, Y 20.1958, Z -5.5000, A 0.000, B 0.000, C 0.000 }
gfCNCPoint4[1633] = {X 181.0813, Y 20.3297, Z -5.5000, A 0.000, B 0.000, C 0.000 }
gfCNCPoint4[1634] = {X 180.8699, Y 21.2784, Z -5.5000, A 0.000, B 0.000, C 0.000 }
gfCNCPoint4[1635] = {X 180.4401, Y 22.1502, Z -5.5000, A 0.000, B 0.000, C 0.000 }
gfCNCPoint4[1636] = {X 179.8163, Y 22.8956, Z -5.5000, A 0.000, B 0.000, C 0.000 }
gfCNCPoint4[1637] = {X 180.1964, Y 22.9068, Z -5.5000, A 0.000, B 0.000, C 0.000 }
gfCNCPoint4[1638] = {X 182.2706, Y 22.6869, Z -5.5000, A 0.000, B 0.000, C 0.000 }
gfCNCPoint4[1639] = {X 184.3520, Y 22.5530, Z -5.5000, A 0.000, B 0.000, C 0.000 }
gfCNCPoint4[1640] = {X 184.7889, Y 22.5370, Z -5.5000, A 0.000, B 0.000, C 0.000 }
gfCNCPoint4[1641] = {X 185.2256, Y 22.5193, Z -5.5000, A 0.000, B 0.000, C 0.000 }
gfCNCPoint4[1642] = {X 189.1921, Y 22.0026, Z -5.5000, A 0.000, B 0.000, C 0.000 }
gfCNCPoint4[1643] = {X 185.1540, Y 22.6024, Z -5.5000, A 0.000, B 0.000, C 0.000 }
gfCNCPoint4[1644] = {X 185.2290, Y 22.5993, Z -5.5000, A 0.000, B 0.000, C 0.000 }
gfCNCPoint4[1645] = {X 187.5635, Y 22.4766, Z -5.5000, A 0.000, B 0.000, C 0.000 }
gfCNCPoint4[1646] = {X 189.8950, Y 22.3063, Z -5.5000, A 0.000, B 0.000, C 0.000 }
gfCNCPoint4[1647] = {X 190.6498, Y 22.2027, Z -5.5000, A 0.000, B 0.000, C 0.000 }
gfCNCPoint4[1648] = {X 191.3815, Y 21.9903, Z -5.5000, A 0.000, B 0.000, C 0.000 }
gfCNCPoint4[1649] = {X 191.4894, Y 21.4334, Z -5.5000, A 0.000, B 0.000, C 0.000 }
gfCNCPoint4[1650] = {X 191.4050, Y 20.8725, Z -5.5000, A 0.000, B 0.000, C 0.000 }
gfCNCPoint4[1651] = {X 191.1380, Y 20.3720, Z -5.5000, A 0.000, B 0.000, C 0.000 }
gfCNCPoint4[1652] = {X 190.7191, Y 19.9895, Z -5.5000, A 0.000, B 0.000, C 0.000 }
gfCNCPoint4[1653] = {X 189.8083, Y 19.5002, Z -5.5000, A 0.000, B 0.000, C 0.000 }
gfCNCPoint4[1654] = {X 188.8335, Y 19.1553, Z -5.5000, A 0.000, B 0.000, C 0.000 }
gfCNCPoint4[1655] = {X 187.8176, Y 18.9629, Z -5.5000, A 0.000, B 0.000, C 0.000 }
gfCNCPoint4[1656] = {X 186.4284, Y 18.8771, Z -5.5000, A 0.000, B 0.000, C 0.000 }
gfCNCPoint4[1657] = {X 185.0380, Y 18.9416, Z -5.5000, A 0.000, B 0.000, C 0.000 }
gfCNCPoint4[1658] = {X 183.6627, Y 19.1556, Z -5.5000, A 0.000, B 0.000, C 0.000 }
gfCNCPoint4[1659] = {X 182.3095, Y 19.5455, Z -5.5000, A 0.000, B 0.000, C 0.000 }
gfCNCPoint4[1660] = {X 181.0351, Y 20.1445, Z -5.5000, A 0.000, B 0.000, C 0.000 }
gfCNCPoint4[1661] = {X 181.0020, Y 20.3183, Z -5.5000, A 0.000, B 0.000, C 0.000 }
gfCNCPoint4[1662] = {X 180.8538, Y 21.0695, Z -5.5000, A 0.000, B 0.000, C 0.000 }
gfCNCPoint4[1663] = {X 180.5651, Y 21.7787, Z -5.5000, A 0.000, B 0.000, C 0.000 }
gfCNCPoint4[1664] = {X 180.1466, Y 22.4199, Z -5.5000, A 0.000, B 0.000, C 0.000 }
gfCNCPoint4[1665] = {X 179.6136, Y 22.9696, Z -5.5000, A 0.000, B 0.000, C 0.000 }
gfCNCPoint4[1666] = {X 180.2003, Y 22.9869, Z -5.5000, A 0.000, B 0.000, C 0.000 }
gfCNCPoint4[1667] = {X 182.2741, Y 22.7669, Z -5.5000, A 0.000, B 0.000, C 0.000 }
gfCNCPoint4[1668] = {X 184.3552, Y 22.6329, Z -5.5000, A 0.000, B 0.000, C 0.000 }
gfCNCPoint4[1669] = {X 184.7921, Y 22.6169, Z -5.5000, A 0.000, B 0.000, C 0.000 }
gfCNCPoint4[1670] = {X 185.2290, Y 22.5993, Z -5.5000, A 0.000, B 0.000, C 0.000 }
gfCNCPoint4[1671] = {X 185.1444, Y 20.6011, Z -5.5000, A 0.000, B 0.000, C 0.000 }
gfCNCPoint4[1672] = {X 185.1444, Y 20.6011, Z -2.5000, A 0.000, B 0.000, C 0.000 }
gfCNCPoint4[1673] = {X 185.1444, Y 20.6011, Z 11.0000, A 0.000, B 0.000, C 0.000 }
gfCNCPoint4[1674] = {X 256.2454, Y 19.7814, Z 11.0000, A 0.000, B 0.000, C 0.000 }
gfCNCPoint4[1675] = {X 256.2454, Y 19.7814, Z -1.6667, A 0.000, B 0.000, C 0.000 }
gfCNCPoint4[1676] = {X 251.5292, Y 19.7814, Z -2.9304, A 0.000, B 0.000, C 0.000 }
gfCNCPoint4[1677] = {X 250.8344, Y 19.7922, Z -3.1166, A 0.000, B 0.000, C 0.000 }
gfCNCPoint4[1678] = {X 250.1815, Y 19.7935, Z -3.2915, A 0.000, B 0.000, C 0.000 }
gfCNCPoint4[1679] = {X 249.4949, Y 19.8921, Z -3.4774, A 0.000, B 0.000, C 0.000 }
gfCNCPoint4[1680] = {X 248.8453, Y 20.0803, Z -3.6586, A 0.000, B 0.000, C 0.000 }
gfCNCPoint4[1681] = {X 248.7084, Y 20.1116, Z -3.6962, A 0.000, B 0.000, C 0.000 }
gfCNCPoint4[1682] = {X 248.6546, Y 20.1622, Z -3.7160, A 0.000, B 0.000, C 0.000 }
gfCNCPoint4[1683] = {X 248.6146, Y 20.2968, Z -3.7536, A 0.000, B 0.000, C 0.000 }
gfCNCPoint4[1684] = {X 248.4756, Y 20.7650, Z -3.8845, A 0.000, B 0.000, C 0.000 }
gfCNCPoint4[1685] = {X 248.4454, Y 21.8671, Z -4.1799, A 0.000, B 0.000, C 0.000 }
gfCNCPoint4[1686] = {X 248.5586, Y 22.3423, Z -4.3108, A 0.000, B 0.000, C 0.000 }
gfCNCPoint4[1687] = {X 248.8748, Y 22.4372, Z -4.3993, A 0.000, B 0.000, C 0.000 }
gfCNCPoint4[1688] = {X 249.2038, Y 22.4643, Z -4.4877, A 0.000, B 0.000, C 0.000 }
gfCNCPoint4[1689] = {X 250.4419, Y 22.5662, Z -4.8206, A 0.000, B 0.000, C 0.000 }
gfCNCPoint4[1690] = {X 251.6873, Y 22.5560, Z -5.1543, A 0.000, B 0.000, C 0.000 }
gfCNCPoint4[1691] = {X 252.9775, Y 22.5560, Z -5.5000, A 0.000, B 0.000, C 0.000 }
gfCNCPoint4[1692] = {X 257.4115, Y 22.5560, Z -5.5000, A 0.000, B 0.000, C 0.000 }
gfCNCPoint4[1693] = {X 257.4115, Y 19.7814, Z -5.5000, A 0.000, B 0.000, C 0.000 }
gfCNCPoint4[1694] = {X 251.5292, Y 19.7814, Z -5.5000, A 0.000, B 0.000, C 0.000 }
gfCNCPoint4[1695] = {X 250.8344, Y 19.7922, Z -5.5000, A 0.000, B 0.000, C 0.000 }
gfCNCPoint4[1696] = {X 249.8296, Y 19.8655, Z -5.5000, A 0.000, B 0.000, C 0.000 }
gfCNCPoint4[1697] = {X 248.8453, Y 20.0803, Z -5.5000, A 0.000, B 0.000, C 0.000 }
gfCNCPoint4[1698] = {X 248.7007, Y 20.1573, Z -5.5000, A 0.000, B 0.000, C 0.000 }
gfCNCPoint4[1699] = {X 248.6146, Y 20.2968, Z -5.5000, A 0.000, B 0.000, C 0.000 }
gfCNCPoint4[1700] = {X 248.4767, Y 20.9719, Z -5.5000, A 0.000, B 0.000, C 0.000 }
gfCNCPoint4[1701] = {X 248.4579, Y 21.6606, Z -5.5000, A 0.000, B 0.000, C 0.000 }
gfCNCPoint4[1702] = {X 248.5586, Y 22.3423, Z -5.5000, A 0.000, B 0.000, C 0.000 }
gfCNCPoint4[1703] = {X 248.8780, Y 22.4202, Z -5.5000, A 0.000, B 0.000, C 0.000 }
gfCNCPoint4[1704] = {X 249.2038, Y 22.4643, Z -5.5000, A 0.000, B 0.000, C 0.000 }
gfCNCPoint4[1705] = {X 250.4445, Y 22.5382, Z -5.5000, A 0.000, B 0.000, C 0.000 }
gfCNCPoint4[1706] = {X 251.6873, Y 22.5560, Z -5.5000, A 0.000, B 0.000, C 0.000 }
gfCNCPoint4[1707] = {X 252.9775, Y 22.5560, Z -5.5000, A 0.000, B 0.000, C 0.000 }
gfCNCPoint4[1708] = {X 248.9927, Y 22.2874, Z -5.5000, A 0.000, B 0.000, C 0.000 }
gfCNCPoint4[1709] = {X 252.9775, Y 22.6360, Z -5.5000, A 0.000, B 0.000, C 0.000 }
gfCNCPoint4[1710] = {X 257.4915, Y 22.6360, Z -5.5000, A 0.000, B 0.000, C 0.000 }
gfCNCPoint4[1711] = {X 257.4915, Y 19.7014, Z -5.5000, A 0.000, B 0.000, C 0.000 }
gfCNCPoint4[1712] = {X 251.5286, Y 19.7014, Z -5.5000, A 0.000, B 0.000, C 0.000 }
gfCNCPoint4[1713] = {X 250.8364, Y 19.7122, Z -5.5000, A 0.000, B 0.000, C 0.000 }
gfCNCPoint4[1714] = {X 249.8259, Y 19.7855, Z -5.5000, A 0.000, B 0.000, C 0.000 }
gfCNCPoint4[1715] = {X 248.8357, Y 20.0005, Z -5.5000, A 0.000, B 0.000, C 0.000 }
gfCNCPoint4[1716] = {X 248.6490, Y 20.0961, Z -5.5000, A 0.000, B 0.000, C 0.000 }
gfCNCPoint4[1717] = {X 248.5379, Y 20.2740, Z -5.5000, A 0.000, B 0.000, C 0.000 }
gfCNCPoint4[1718] = {X 248.3955, Y 20.9779, Z -5.5000, A 0.000, B 0.000, C 0.000 }
gfCNCPoint4[1719] = {X 248.3799, Y 21.6959, Z -5.5000, A 0.000, B 0.000, C 0.000 }
gfCNCPoint4[1720] = {X 248.4917, Y 22.4053, Z -5.5000, A 0.000, B 0.000, C 0.000 }
gfCNCPoint4[1721] = {X 248.8406, Y 22.4945, Z -5.5000, A 0.000, B 0.000, C 0.000 }
gfCNCPoint4[1722] = {X 249.1972, Y 22.5440, Z -5.5000, A 0.000, B 0.000, C 0.000 }
gfCNCPoint4[1723] = {X 250.4406, Y 22.6181, Z -5.5000, A 0.000, B 0.000, C 0.000 }
gfCNCPoint4[1724] = {X 251.6860, Y 22.6360, Z -5.5000, A 0.000, B 0.000, C 0.000 }
gfCNCPoint4[1725] = {X 252.9775, Y 22.6360, Z -5.5000, A 0.000, B 0.000, C 0.000 }
gfCNCPoint4[1726] = {X 256.9623, Y 22.2874, Z -5.5000, A 0.000, B 0.000, C 0.000 }
gfCNCPoint4[1727] = {X 248.9927, Y 22.3674, Z -5.5000, A 0.000, B 0.000, C 0.000 }
gfCNCPoint4[1728] = {X 252.9775, Y 22.7160, Z -5.5000, A 0.000, B 0.000, C 0.000 }
gfCNCPoint4[1729] = {X 257.5715, Y 22.7160, Z -5.5000, A 0.000, B 0.000, C 0.000 }
gfCNCPoint4[1730] = {X 257.5715, Y 19.6214, Z -5.5000, A 0.000, B 0.000, C 0.000 }
gfCNCPoint4[1731] = {X 251.5280, Y 19.6214, Z -5.5000, A 0.000, B 0.000, C 0.000 }
gfCNCPoint4[1732] = {X 250.8357, Y 19.6322, Z -5.5000, A 0.000, B 0.000, C 0.000 }
gfCNCPoint4[1733] = {X 249.8156, Y 19.7062, Z -5.5000, A 0.000, B 0.000, C 0.000 }
gfCNCPoint4[1734] = {X 248.8161, Y 19.9229, Z -5.5000, A 0.000, B 0.000, C 0.000 }
gfCNCPoint4[1735] = {X 248.5936, Y 20.0384, Z -5.5000, A 0.000, B 0.000, C 0.000 }
gfCNCPoint4[1736] = {X 248.4612, Y 20.2512, Z -5.5000, A 0.000, B 0.000, C 0.000 }
gfCNCPoint4[1737] = {X 248.3144, Y 20.9838, Z -5.5000, A 0.000, B 0.000, C 0.000 }
gfCNCPoint4[1738] = {X 248.3022, Y 21.7309, Z -5.5000, A 0.000, B 0.000, C 0.000 }
gfCNCPoint4[1739] = {X 248.4251, Y 22.4679, Z -5.5000, A 0.000, B 0.000, C 0.000 }
gfCNCPoint4[1740] = {X 248.8033, Y 22.5686, Z -5.5000, A 0.000, B 0.000, C 0.000 }
gfCNCPoint4[1741] = {X 249.1906, Y 22.6238, Z -5.5000, A 0.000, B 0.000, C 0.000 }
gfCNCPoint4[1742] = {X 250.4375, Y 22.6981, Z -5.5000, A 0.000, B 0.000, C 0.000 }
gfCNCPoint4[1743] = {X 251.6864, Y 22.7160, Z -5.5000, A 0.000, B 0.000, C 0.000 }
gfCNCPoint4[1744] = {X 252.9775, Y 22.7160, Z -5.5000, A 0.000, B 0.000, C 0.000 }
gfCNCPoint4[1745] = {X 256.9623, Y 22.3674, Z -5.5000, A 0.000, B 0.000, C 0.000 }
gfCNCPoint4[1746] = {X 248.9927, Y 22.4474, Z -5.5000, A 0.000, B 0.000, C 0.000 }
gfCNCPoint4[1747] = {X 252.9775, Y 22.7960, Z -5.5000, A 0.000, B 0.000, C 0.000 }
gfCNCPoint4[1748] = {X 257.6515, Y 22.7960, Z -5.5000, A 0.000, B 0.000, C 0.000 }
gfCNCPoint4[1749] = {X 257.6515, Y 19.5414, Z -5.5000, A 0.000, B 0.000, C 0.000 }
gfCNCPoint4[1750] = {X 251.5274, Y 19.5414, Z -5.5000, A 0.000, B 0.000, C 0.000 }
gfCNCPoint4[1751] = {X 250.8350, Y 19.5522, Z -5.5000, A 0.000, B 0.000, C 0.000 }
gfCNCPoint4[1752] = {X 249.8053, Y 19.6268, Z -5.5000, A 0.000, B 0.000, C 0.000 }
gfCNCPoint4[1753] = {X 248.7963, Y 19.8454, Z -5.5000, A 0.000, B 0.000, C 0.000 }
gfCNCPoint4[1754] = {X 248.5381, Y 19.9807, Z -5.5000, A 0.000, B 0.000, C 0.000 }
gfCNCPoint4[1755] = {X 248.3845, Y 20.2285, Z -5.5000, A 0.000, B 0.000, C 0.000 }
gfCNCPoint4[1756] = {X 248.2333, Y 20.9896, Z -5.5000, A 0.000, B 0.000, C 0.000 }
gfCNCPoint4[1757] = {X 248.2247, Y 21.7656, Z -5.5000, A 0.000, B 0.000, C 0.000 }
gfCNCPoint4[1758] = {X 248.3589, Y 22.5299, Z -5.5000, A 0.000, B 0.000, C 0.000 }
gfCNCPoint4[1759] = {X 248.7661, Y 22.6426, Z -5.5000, A 0.000, B 0.000, C 0.000 }
gfCNCPoint4[1760] = {X 249.1841, Y 22.7035, Z -5.5000, A 0.000, B 0.000, C 0.000 }
gfCNCPoint4[1761] = {X 250.4343, Y 22.7780, Z -5.5000, A 0.000, B 0.000, C 0.000 }
gfCNCPoint4[1762] = {X 251.6867, Y 22.7960, Z -5.5000, A 0.000, B 0.000, C 0.000 }
gfCNCPoint4[1763] = {X 252.9775, Y 22.7960, Z -5.5000, A 0.000, B 0.000, C 0.000 }
gfCNCPoint4[1764] = {X 256.9623, Y 22.4474, Z -5.5000, A 0.000, B 0.000, C 0.000 }
gfCNCPoint4[1765] = {X 248.9927, Y 22.5274, Z -5.5000, A 0.000, B 0.000, C 0.000 }
gfCNCPoint4[1766] = {X 252.9775, Y 22.8760, Z -5.5000, A 0.000, B 0.000, C 0.000 }
gfCNCPoint4[1767] = {X 257.7315, Y 22.8760, Z -5.5000, A 0.000, B 0.000, C 0.000 }
gfCNCPoint4[1768] = {X 257.7315, Y 19.4614, Z -5.5000, A 0.000, B 0.000, C 0.000 }
gfCNCPoint4[1769] = {X 251.5267, Y 19.4614, Z -5.5000, A 0.000, B 0.000, C 0.000 }
gfCNCPoint4[1770] = {X 250.8343, Y 19.4722, Z -5.5000, A 0.000, B 0.000, C 0.000 }
gfCNCPoint4[1771] = {X 249.7949, Y 19.5475, Z -5.5000, A 0.000, B 0.000, C 0.000 }
gfCNCPoint4[1772] = {X 248.7763, Y 19.7679, Z -5.5000, A 0.000, B 0.000, C 0.000 }
gfCNCPoint4[1773] = {X 248.4826, Y 19.9231, Z -5.5000, A 0.000, B 0.000, C 0.000 }
gfCNCPoint4[1774] = {X 248.3078, Y 20.2057, Z -5.5000, A 0.000, B 0.000, C 0.000 }
gfCNCPoint4[1775] = {X 248.1530, Y 20.9889, Z -5.5000, A 0.000, B 0.000, C 0.000 }
gfCNCPoint4[1776] = {X 248.1462, Y 21.7872, Z -5.5000, A 0.000, B 0.000, C 0.000 }
gfCNCPoint4[1777] = {X 248.2878, Y 22.5729, Z -5.5000, A 0.000, B 0.000, C 0.000 }
gfCNCPoint4[1778] = {X 248.3065, Y 22.5963, Z -5.5000, A 0.000, B 0.000, C 0.000 }
gfCNCPoint4[1779] = {X 248.3328, Y 22.6055, Z -5.5000, A 0.000, B 0.000, C 0.000 }
gfCNCPoint4[1780] = {X 248.7496, Y 22.7209, Z -5.5000, A 0.000, B 0.000, C 0.000 }
gfCNCPoint4[1781] = {X 249.1775, Y 22.7832, Z -5.5000, A 0.000, B 0.000, C 0.000 }
gfCNCPoint4[1782] = {X 250.4312, Y 22.8580, Z -5.5000, A 0.000, B 0.000, C 0.000 }
gfCNCPoint4[1783] = {X 251.6870, Y 22.8760, Z -5.5000, A 0.000, B 0.000, C 0.000 }
gfCNCPoint4[1784] = {X 252.9775, Y 22.8760, Z -5.5000, A 0.000, B 0.000, C 0.000 }
gfCNCPoint4[1785] = {X 256.9623, Y 22.5274, Z -5.5000, A 0.000, B 0.000, C 0.000 }
gfCNCPoint4[1786] = {X 248.9927, Y 22.6074, Z -5.5000, A 0.000, B 0.000, C 0.000 }
gfCNCPoint4[1787] = {X 252.9775, Y 22.9560, Z -5.5000, A 0.000, B 0.000, C 0.000 }
gfCNCPoint4[1788] = {X 257.8115, Y 22.9560, Z -5.5000, A 0.000, B 0.000, C 0.000 }
gfCNCPoint4[1789] = {X 257.8113, Y 19.3814, Z -5.5000, A 0.000, B 0.000, C 0.000 }
gfCNCPoint4[1790] = {X 251.5261, Y 19.3814, Z -5.5000, A 0.000, B 0.000, C 0.000 }
gfCNCPoint4[1791] = {X 250.8336, Y 19.3922, Z -5.5000, A 0.000, B 0.000, C 0.000 }
gfCNCPoint4[1792] = {X 249.7844, Y 19.4682, Z -5.5000, A 0.000, B 0.000, C 0.000 }
gfCNCPoint4[1793] = {X 248.7562, Y 19.6904, Z -5.5000, A 0.000, B 0.000, C 0.000 }
gfCNCPoint4[1794] = {X 248.4270, Y 19.8656, Z -5.5000, A 0.000, B 0.000, C 0.000 }
gfCNCPoint4[1795] = {X 248.2311, Y 20.1829, Z -5.5000, A 0.000, B 0.000, C 0.000 }
gfCNCPoint4[1796] = {X 248.0728, Y 20.9862, Z -5.5000, A 0.000, B 0.000, C 0.000 }
gfCNCPoint4[1797] = {X 248.0674, Y 21.8049, Z -5.5000, A 0.000, B 0.000, C 0.000 }
gfCNCPoint4[1798] = {X 248.2151, Y 22.6102, Z -5.5000, A 0.000, B 0.000, C 0.000 }
gfCNCPoint4[1799] = {X 248.2581, Y 22.6640, Z -5.5000, A 0.000, B 0.000, C 0.000 }
gfCNCPoint4[1800] = {X 248.7079, Y 22.7938, Z -5.5000, A 0.000, B 0.000, C 0.000 }
gfCNCPoint4[1801] = {X 249.1710, Y 22.8630, Z -5.5000, A 0.000, B 0.000, C 0.000 }
gfCNCPoint4[1802] = {X 250.4281, Y 22.9379, Z -5.5000, A 0.000, B 0.000, C 0.000 }
gfCNCPoint4[1803] = {X 251.6873, Y 22.9560, Z -5.5000, A 0.000, B 0.000, C 0.000 }
gfCNCPoint4[1804] = {X 252.9775, Y 22.9560, Z -5.5000, A 0.000, B 0.000, C 0.000 }
gfCNCPoint4[1805] = {X 256.9623, Y 22.6074, Z -5.5000, A 0.000, B 0.000, C 0.000 }
gfCNCPoint4[1806] = {X 256.9623, Y 22.6074, Z -2.5000, A 0.000, B 0.000, C 0.000 }
gfCNCPoint4[1807] = {X 256.9623, Y 22.6074, Z 11.0000, A 0.000, B 0.000, C 0.000 }
gfCNCPoint4[1808] = {X 507.6814, Y 107.6951, Z 11.0000, A 0.000, B 0.000, C 0.000 }
gfCNCPoint4[1809] = {X 507.6814, Y 107.6951, Z -2.5000, A 0.000, B 0.000, C 0.000 }
gfCNCPoint4[1810] = {X 507.6814, Y 107.6951, Z -5.5000, A 0.000, B 0.000, C 0.000 }
gfCNCPoint4[1811] = {X 507.6814, Y 71.2951, Z -5.5000, A 0.000, B 0.000, C 0.000 }
gfCNCPoint4[1812] = {X 509.5503, Y 71.2951, Z -5.5000, A 0.000, B 0.000, C 0.000 }
gfCNCPoint4[1813] = {X 509.0279, Y 71.0691, Z -5.5000, A 0.000, B 0.000, C 0.000 }
gfCNCPoint4[1814] = {X 508.5105, Y 70.8320, Z -5.5000, A 0.000, B 0.000, C 0.000 }
gfCNCPoint4[1815] = {X 507.1675, Y 71.0984, Z -5.5000, A 0.000, B 0.000, C 0.000 }
gfCNCPoint4[1816] = {X 505.8126, Y 71.2951, Z -5.5000, A 0.000, B 0.000, C 0.000 }
gfCNCPoint4[1817] = {X 507.6814, Y 71.2951, Z -5.5000, A 0.000, B 0.000, C 0.000 }
gfCNCPoint4[1818] = {X 507.6814, Y 73.6951, Z -5.5000, A 0.000, B 0.000, C 0.000 }
gfCNCPoint4[1819] = {X 551.2535, Y 73.6951, Z -5.5000, A 0.000, B 0.000, C 0.000 }
gfCNCPoint4[1820] = {X 549.1240, Y 72.7707, Z -5.5000, A 0.000, B 0.000, C 0.000 }
gfCNCPoint4[1821] = {X 547.0701, Y 71.6885, Z -5.5000, A 0.000, B 0.000, C 0.000 }
gfCNCPoint4[1822] = {X 545.1036, Y 70.4547, Z -5.5000, A 0.000, B 0.000, C 0.000 }
gfCNCPoint4[1823] = {X 543.2356, Y 69.0763, Z -5.5000, A 0.000, B 0.000, C 0.000 }
gfCNCPoint4[1824] = {X 529.7631, Y 69.0765, Z -5.5000, A 0.000, B 0.000, C 0.000 }
gfCNCPoint4[1825] = {X 527.5580, Y 69.8774, Z -5.5000, A 0.000, B 0.000, C 0.000 }
gfCNCPoint4[1826] = {X 525.2858, Y 70.4613, Z -5.5000, A 0.000, B 0.000, C 0.000 }
gfCNCPoint4[1827] = {X 522.9678, Y 70.8229, Z -5.5000, A 0.000, B 0.000, C 0.000 }
gfCNCPoint4[1828] = {X 520.6258, Y 70.9586, Z -5.5000, A 0.000, B 0.000, C 0.000 }
gfCNCPoint4[1829] = {X 519.7998, Y 70.9591, Z -5.5000, A 0.000, B 0.000, C 0.000 }
gfCNCPoint4[1830] = {X 517.4111, Y 70.8403, Z -5.5000, A 0.000, B 0.000, C 0.000 }
gfCNCPoint4[1831] = {X 515.0460, Y 70.4852, Z -5.5000, A 0.000, B 0.000, C 0.000 }
gfCNCPoint4[1832] = {X 512.7277, Y 69.8972, Z -5.5000, A 0.000, B 0.000, C 0.000 }
gfCNCPoint4[1833] = {X 510.4792, Y 69.0821, Z -5.5000, A 0.000, B 0.000, C 0.000 }
gfCNCPoint4[1834] = {X 509.6266, Y 68.7046, Z -5.5000, A 0.000, B 0.000, C 0.000 }
gfCNCPoint4[1835] = {X 508.7892, Y 68.2944, Z -5.5000, A 0.000, B 0.000, C 0.000 }
gfCNCPoint4[1836] = {X 507.1699, Y 68.6593, Z -5.5000, A 0.000, B 0.000, C 0.000 }
gfCNCPoint4[1837] = {X 505.5294, Y 68.9118, Z -5.5000, A 0.000, B 0.000, C 0.000 }
gfCNCPoint4[1838] = {X 504.1114, Y 69.0379, Z -5.5000, A 0.000, B 0.000, C 0.000 }
gfCNCPoint4[1839] = {X 502.6885, Y 69.0800, Z -5.5000, A 0.000, B 0.000, C 0.000 }
gfCNCPoint4[1840] = {X 502.0391, Y 69.0800, Z -5.5000, A 0.000, B 0.000, C 0.000 }
gfCNCPoint4[1841] = {X 501.1776, Y 71.1319, Z -5.5000, A 0.000, B 0.000, C 0.000 }
gfCNCPoint4[1842] = {X 500.1606, Y 73.1114, Z -5.5000, A 0.000, B 0.000, C 0.000 }
gfCNCPoint4[1843] = {X 500.1606, Y 73.6951, Z -5.5000, A 0.000, B 0.000, C 0.000 }
gfCNCPoint4[1844] = {X 507.6814, Y 73.6951, Z -5.5000, A 0.000, B 0.000, C 0.000 }
gfCNCPoint4[1845] = {X 507.6814, Y 76.0951, Z -5.5000, A 0.000, B 0.000, C 0.000 }
gfCNCPoint4[1846] = {X 576.0966, Y 76.0951, Z -5.5000, A 0.000, B 0.000, C 0.000 }
gfCNCPoint4[1847] = {X 576.0966, Y 72.8901, Z -5.5000, A 0.000, B 0.000, C 0.000 }
gfCNCPoint4[1848] = {X 575.7178, Y 72.8147, Z -5.5000, A 0.000, B 0.000, C 0.000 }
gfCNCPoint4[1849] = {X 575.3401, Y 72.7341, Z -5.5000, A 0.000, B 0.000, C 0.000 }
gfCNCPoint4[1850] = {X 573.3201, Y 73.1034, Z -5.5000, A 0.000, B 0.000, C 0.000 }
gfCNCPoint4[1851] = {X 571.2786, Y 73.3258, Z -5.5000, A 0.000, B 0.000, C 0.000 }
gfCNCPoint4[1852] = {X 569.2264, Y 73.4000, Z -5.5000, A 0.000, B 0.000, C 0.000 }
gfCNCPoint4[1853] = {X 562.4443, Y 73.4000, Z -5.5000, A 0.000, B 0.000, C 0.000 }
gfCNCPoint4[1854] = {X 560.3342, Y 73.3215, Z -5.5000, A 0.000, B 0.000, C 0.000 }
gfCNCPoint4[1855] = {X 558.2357, Y 73.0864, Z -5.5000, A 0.000, B 0.000, C 0.000 }
gfCNCPoint4[1856] = {X 556.1605, Y 72.6961, Z -5.5000, A 0.000, B 0.000, C 0.000 }
gfCNCPoint4[1857] = {X 554.1200, Y 72.1526, Z -5.5000, A 0.000, B 0.000, C 0.000 }
gfCNCPoint4[1858] = {X 552.1255, Y 71.4591, Z -5.5000, A 0.000, B 0.000, C 0.000 }
gfCNCPoint4[1859] = {X 549.9764, Y 70.5169, Z -5.5000, A 0.000, B 0.000, C 0.000 }
gfCNCPoint4[1860] = {X 547.9124, Y 69.4005, Z -5.5000, A 0.000, B 0.000, C 0.000 }
gfCNCPoint4[1861] = {X 545.9476, Y 68.1175, Z -5.5000, A 0.000, B 0.000, C 0.000 }
gfCNCPoint4[1862] = {X 544.0954, Y 66.6766, Z -5.5000, A 0.000, B 0.000, C 0.000 }
gfCNCPoint4[1863] = {X 543.8502, Y 66.6778, Z -5.5000, A 0.000, B 0.000, C 0.000 }
gfCNCPoint4[1864] = {X 543.6050, Y 66.6763, Z -5.5000, A 0.000, B 0.000, C 0.000 }
gfCNCPoint4[1865] = {X 529.2675, Y 66.6766, Z -5.5000, A 0.000, B 0.000, C 0.000 }
gfCNCPoint4[1866] = {X 527.1875, Y 67.4768, Z -5.5000, A 0.000, B 0.000, C 0.000 }
gfCNCPoint4[1867] = {X 525.0367, Y 68.0609, Z -5.5000, A 0.000, B 0.000, C 0.000 }
gfCNCPoint4[1868] = {X 522.8376, Y 68.4228, Z -5.5000, A 0.000, B 0.000, C 0.000 }
gfCNCPoint4[1869] = {X 520.6131, Y 68.5586, Z -5.5000, A 0.000, B 0.000, C 0.000 }
gfCNCPoint4[1870] = {X 519.7998, Y 68.5591, Z -5.5000, A 0.000, B 0.000, C 0.000 }
gfCNCPoint4[1871] = {X 517.5593, Y 68.4430, Z -5.5000, A 0.000, B 0.000, C 0.000 }
gfCNCPoint4[1872] = {X 515.3429, Y 68.0961, Z -5.5000, A 0.000, B 0.000, C 0.000 }
gfCNCPoint4[1873] = {X 513.1742, Y 67.5219, Z -5.5000, A 0.000, B 0.000, C 0.000 }
gfCNCPoint4[1874] = {X 511.0764, Y 66.7267, Z -5.5000, A 0.000, B 0.000, C 0.000 }
gfCNCPoint4[1875] = {X 509.0720, Y 65.7189, Z -5.5000, A 0.000, B 0.000, C 0.000 }
gfCNCPoint4[1876] = {X 506.9797, Y 66.2511, Z -5.5000, A 0.000, B 0.000, C 0.000 }
gfCNCPoint4[1877] = {X 504.8448, Y 66.5725, Z -5.5000, A 0.000, B 0.000, C 0.000 }
gfCNCPoint4[1878] = {X 502.6885, Y 66.6800, Z -5.5000, A 0.000, B 0.000, C 0.000 }
gfCNCPoint4[1879] = {X 500.3217, Y 66.6800, Z -5.5000, A 0.000, B 0.000, C 0.000 }
gfCNCPoint4[1880] = {X 499.6232, Y 68.6752, Z -5.5000, A 0.000, B 0.000, C 0.000 }
gfCNCPoint4[1881] = {X 498.7676, Y 70.6084, Z -5.5000, A 0.000, B 0.000, C 0.000 }
gfCNCPoint4[1882] = {X 497.7606, Y 72.4672, Z -5.5000, A 0.000, B 0.000, C 0.000 }
gfCNCPoint4[1883] = {X 497.7607, Y 76.0951, Z -5.5000, A 0.000, B 0.000, C 0.000 }
gfCNCPoint4[1884] = {X 507.6814, Y 76.0951, Z -5.5000, A 0.000, B 0.000, C 0.000 }
gfCNCPoint4[1885] = {X 507.6814, Y 78.4951, Z -5.5000, A 0.000, B 0.000, C 0.000 }
gfCNCPoint4[1886] = {X 578.4966, Y 78.4951, Z -5.5000, A 0.000, B 0.000, C 0.000 }
gfCNCPoint4[1887] = {X 578.4966, Y 70.8313, Z -5.5000, A 0.000, B 0.000, C 0.000 }
gfCNCPoint4[1888] = {X 576.9097, Y 70.5998, Z -5.5000, A 0.000, B 0.000, C 0.000 }
gfCNCPoint4[1889] = {X 575.3401, Y 70.2710, Z -5.5000, A 0.000, B 0.000, C 0.000 }
gfCNCPoint4[1890] = {X 573.3236, Y 70.6751, Z -5.5000, A 0.000, B 0.000, C 0.000 }
gfCNCPoint4[1891] = {X 571.2815, Y 70.9187, Z -5.5000, A 0.000, B 0.000, C 0.000 }
gfCNCPoint4[1892] = {X 569.2264, Y 71.0000, Z -5.5000, A 0.000, B 0.000, C 0.000 }
gfCNCPoint4[1893] = {X 562.4443, Y 71.0000, Z -5.5000, A 0.000, B 0.000, C 0.000 }
gfCNCPoint4[1894] = {X 560.0513, Y 70.8896, Z -5.5000, A 0.000, B 0.000, C 0.000 }
gfCNCPoint4[1895] = {X 557.6786, Y 70.5595, Z -5.5000, A 0.000, B 0.000, C 0.000 }
gfCNCPoint4[1896] = {X 555.3464, Y 70.0124, Z -5.5000, A 0.000, B 0.000, C 0.000 }
gfCNCPoint4[1897] = {X 553.0745, Y 69.2530, Z -5.5000, A 0.000, B 0.000, C 0.000 }
gfCNCPoint4[1898] = {X 550.8820, Y 68.2876, Z -5.5000, A 0.000, B 0.000, C 0.000 }
gfCNCPoint4[1899] = {X 548.7878, Y 67.1246, Z -5.5000, A 0.000, B 0.000, C 0.000 }
gfCNCPoint4[1900] = {X 546.8094, Y 65.7738, Z -5.5000, A 0.000, B 0.000, C 0.000 }
gfCNCPoint4[1901] = {X 544.9638, Y 64.2466, Z -5.5000, A 0.000, B 0.000, C 0.000 }
gfCNCPoint4[1902] = {X 544.2921, Y 64.2732, Z -5.5000, A 0.000, B 0.000, C 0.000 }
gfCNCPoint4[1903] = {X 543.6199, Y 64.2763, Z -5.5000, A 0.000, B 0.000, C 0.000 }
gfCNCPoint4[1904] = {X 528.7425, Y 64.2766, Z -5.5000, A 0.000, B 0.000, C 0.000 }
gfCNCPoint4[1905] = {X 526.7929, Y 65.0770, Z -5.5000, A 0.000, B 0.000, C 0.000 }
gfCNCPoint4[1906] = {X 524.7682, Y 65.6616, Z -5.5000, A 0.000, B 0.000, C 0.000 }
gfCNCPoint4[1907] = {X 522.6921, Y 66.0236, Z -5.5000, A 0.000, B 0.000, C 0.000 }
gfCNCPoint4[1908] = {X 520.5890, Y 66.1587, Z -5.5000, A 0.000, B 0.000, C 0.000 }
gfCNCPoint4[1909] = {X 519.7998, Y 66.1591, Z -5.5000, A 0.000, B 0.000, C 0.000 }
gfCNCPoint4[1910] = {X 517.9641, Y 66.0715, Z -5.5000, A 0.000, B 0.000, C 0.000 }
gfCNCPoint4[1911] = {X 516.1450, Y 65.8096, Z -5.5000, A 0.000, B 0.000, C 0.000 }
gfCNCPoint4[1912] = {X 514.3592, Y 65.3756, Z -5.5000, A 0.000, B 0.000, C 0.000 }
gfCNCPoint4[1913] = {X 512.6228, Y 64.7735, Z -5.5000, A 0.000, B 0.000, C 0.000 }
gfCNCPoint4[1914] = {X 510.9516, Y 64.0089, Z -5.5000, A 0.000, B 0.000, C 0.000 }
gfCNCPoint4[1915] = {X 509.3609, Y 63.0886, Z -5.5000, A 0.000, B 0.000, C 0.000 }
gfCNCPoint4[1916] = {X 507.7389, Y 63.6068, Z -5.5000, A 0.000, B 0.000, C 0.000 }
gfCNCPoint4[1917] = {X 506.0774, Y 63.9798, Z -5.5000, A 0.000, B 0.000, C 0.000 }
gfCNCPoint4[1918] = {X 504.3896, Y 64.2048, Z -5.5000, A 0.000, B 0.000, C 0.000 }
gfCNCPoint4[1919] = {X 502.6885, Y 64.2800, Z -5.5000, A 0.000, B 0.000, C 0.000 }
gfCNCPoint4[1920] = {X 498.4791, Y 64.2800, Z -5.5000, A 0.000, B 0.000, C 0.000 }
gfCNCPoint4[1921] = {X 497.9417, Y 66.2503, Z -5.5000, A 0.000, B 0.000, C 0.000 }
gfCNCPoint4[1922] = {X 497.2392, Y 68.1679, Z -5.5000, A 0.000, B 0.000, C 0.000 }
gfCNCPoint4[1923] = {X 496.3768, Y 70.0192, Z -5.5000, A 0.000, B 0.000, C 0.000 }
gfCNCPoint4[1924] = {X 495.3606, Y 71.7907, Z -5.5000, A 0.000, B 0.000, C 0.000 }
gfCNCPoint4[1925] = {X 495.3607, Y 78.4951, Z -5.5000, A 0.000, B 0.000, C 0.000 }
gfCNCPoint4[1926] = {X 507.6814, Y 78.4951, Z -5.5000, A 0.000, B 0.000, C 0.000 }
gfCNCPoint4[1927] = {X 507.6814, Y 80.8951, Z -5.5000, A 0.000, B 0.000, C 0.000 }
gfCNCPoint4[1928] = {X 580.8966, Y 80.8951, Z -5.5000, A 0.000, B 0.000, C 0.000 }
gfCNCPoint4[1929] = {X 580.8966, Y 68.5934, Z -5.5000, A 0.000, B 0.000, C 0.000 }
gfCNCPoint4[1930] = {X 579.0252, Y 68.4747, Z -5.5000, A 0.000, B 0.000, C 0.000 }
gfCNCPoint4[1931] = {X 577.1692, Y 68.2078, Z -5.5000, A 0.000, B 0.000, C 0.000 }
gfCNCPoint4[1932] = {X 575.3401, Y 67.7943, Z -5.5000, A 0.000, B 0.000, C 0.000 }
gfCNCPoint4[1933] = {X 573.3283, Y 68.2408, Z -5.5000, A 0.000, B 0.000, C 0.000 }
gfCNCPoint4[1934] = {X 571.2852, Y 68.5100, Z -5.5000, A 0.000, B 0.000, C 0.000 }
gfCNCPoint4[1935] = {X 569.2264, Y 68.6000, Z -5.5000, A 0.000, B 0.000, C 0.000 }
gfCNCPoint4[1936] = {X 562.4443, Y 68.6000, Z -5.5000, A 0.000, B 0.000, C 0.000 }
gfCNCPoint4[1937] = {X 560.1444, Y 68.4877, Z -5.5000, A 0.000, B 0.000, C 0.000 }
gfCNCPoint4[1938] = {X 557.8664, Y 68.1517, Z -5.5000, A 0.000, B 0.000, C 0.000 }
gfCNCPoint4[1939] = {X 555.6319, Y 67.5954, Z -5.5000, A 0.000, B 0.000, C 0.000 }
gfCNCPoint4[1940] = {X 553.4623, Y 66.8239, Z -5.5000, A 0.000, B 0.000, C 0.000 }
gfCNCPoint4[1941] = {X 551.3783, Y 65.8447, Z -5.5000, A 0.000, B 0.000, C 0.000 }
gfCNCPoint4[1942] = {X 549.3995, Y 64.6671, Z -5.5000, A 0.000, B 0.000, C 0.000 }
gfCNCPoint4[1943] = {X 547.5450, Y 63.3022, Z -5.5000, A 0.000, B 0.000, C 0.000 }
gfCNCPoint4[1944] = {X 545.8323, Y 61.7631, Z -5.5000, A 0.000, B 0.000, C 0.000 }
gfCNCPoint4[1945] = {X 544.7359, Y 61.8555, Z -5.5000, A 0.000, B 0.000, C 0.000 }
gfCNCPoint4[1946] = {X 543.6357, Y 61.8763, Z -5.5000, A 0.000, B 0.000, C 0.000 }
gfCNCPoint4[1947] = {X 528.1821, Y 61.8766, Z -5.5000, A 0.000, B 0.000, C 0.000 }
gfCNCPoint4[1948] = {X 526.3756, Y 62.6760, Z -5.5000, A 0.000, B 0.000, C 0.000 }
gfCNCPoint4[1949] = {X 524.4886, Y 63.2609, Z -5.5000, A 0.000, B 0.000, C 0.000 }
gfCNCPoint4[1950] = {X 522.5466, Y 63.6234, Z -5.5000, A 0.000, B 0.000, C 0.000 }
gfCNCPoint4[1951] = {X 520.5757, Y 63.7587, Z -5.5000, A 0.000, B 0.000, C 0.000 }
gfCNCPoint4[1952] = {X 519.7998, Y 63.7591, Z -5.5000, A 0.000, B 0.000, C 0.000 }
gfCNCPoint4[1953] = {X 517.9902, Y 63.6618, Z -5.5000, A 0.000, B 0.000, C 0.000 }
gfCNCPoint4[1954] = {X 516.2015, Y 63.3711, Z -5.5000, A 0.000, B 0.000, C 0.000 }
gfCNCPoint4[1955] = {X 514.4543, Y 62.8904, Z -5.5000, A 0.000, B 0.000, C 0.000 }
gfCNCPoint4[1956] = {X 512.7687, Y 62.2251, Z -5.5000, A 0.000, B 0.000, C 0.000 }
gfCNCPoint4[1957] = {X 511.1641, Y 61.3829, Z -5.5000, A 0.000, B 0.000, C 0.000 }
gfCNCPoint4[1958] = {X 509.6590, Y 60.3735, Z -5.5000, A 0.000, B 0.000, C 0.000 }
gfCNCPoint4[1959] = {X 507.9866, Y 61.0270, Z -5.5000, A 0.000, B 0.000, C 0.000 }
gfCNCPoint4[1960] = {X 506.2542, Y 61.4991, Z -5.5000, A 0.000, B 0.000, C 0.000 }
gfCNCPoint4[1961] = {X 504.4815, Y 61.7845, Z -5.5000, A 0.000, B 0.000, C 0.000 }
gfCNCPoint4[1962] = {X 502.6885, Y 61.8800, Z -5.5000, A 0.000, B 0.000, C 0.000 }
gfCNCPoint4[1963] = {X 496.4789, Y 61.8800, Z -5.5000, A 0.000, B 0.000, C 0.000 }
gfCNCPoint4[1964] = {X 496.1192, Y 63.8331, Z -5.5000, A 0.000, B 0.000, C 0.000 }
gfCNCPoint4[1965] = {X 495.5823, Y 65.7451, Z -5.5000, A 0.000, B 0.000, C 0.000 }
gfCNCPoint4[1966] = {X 494.8727, Y 67.5999, Z -5.5000, A 0.000, B 0.000, C 0.000 }
gfCNCPoint4[1967] = {X 493.9964, Y 69.3821, Z -5.5000, A 0.000, B 0.000, C 0.000 }
gfCNCPoint4[1968] = {X 492.9606, Y 71.0765, Z -5.5000, A 0.000, B 0.000, C 0.000 }
gfCNCPoint4[1969] = {X 492.9607, Y 80.8951, Z -5.5000, A 0.000, B 0.000, C 0.000 }
gfCNCPoint4[1970] = {X 507.6814, Y 80.8951, Z -5.5000, A 0.000, B 0.000, C 0.000 }
gfCNCPoint4[1971] = {X 507.6814, Y 83.2951, Z -5.5000, A 0.000, B 0.000, C 0.000 }
gfCNCPoint4[1972] = {X 583.2966, Y 83.2951, Z -5.5000, A 0.000, B 0.000, C 0.000 }
gfCNCPoint4[1973] = {X 583.2966, Y 66.1198, Z -5.5000, A 0.000, B 0.000, C 0.000 }
gfCNCPoint4[1974] = {X 581.2872, Y 66.1993, Z -5.5000, A 0.000, B 0.000, C 0.000 }
gfCNCPoint4[1975] = {X 579.2793, Y 66.0882, Z -5.5000, A 0.000, B 0.000, C 0.000 }
gfCNCPoint4[1976] = {X 577.2910, Y 65.7873, Z -5.5000, A 0.000, B 0.000, C 0.000 }
gfCNCPoint4[1977] = {X 575.3401, Y 65.2993, Z -5.5000, A 0.000, B 0.000, C 0.000 }
gfCNCPoint4[1978] = {X 573.3348, Y 65.7981, Z -5.5000, A 0.000, B 0.000, C 0.000 }
gfCNCPoint4[1979] = {X 571.2904, Y 66.0993, Z -5.5000, A 0.000, B 0.000, C 0.000 }
gfCNCPoint4[1980] = {X 569.2264, Y 66.2000, Z -5.5000, A 0.000, B 0.000, C 0.000 }
gfCNCPoint4[1981] = {X 562.4443, Y 66.2000, Z -5.5000, A 0.000, B 0.000, C 0.000 }
gfCNCPoint4[1982] = {X 560.2304, Y 66.0841, Z -5.5000, A 0.000, B 0.000, C 0.000 }
gfCNCPoint4[1983] = {X 558.0406, Y 65.7376, Z -5.5000, A 0.000, B 0.000, C 0.000 }
gfCNCPoint4[1984] = {X 555.8991, Y 65.1643, Z -5.5000, A 0.000, B 0.000, C 0.000 }
gfCNCPoint4[1985] = {X 553.8291, Y 64.3705, Z -5.5000, A 0.000, B 0.000, C 0.000 }
gfCNCPoint4[1986] = {X 551.8533, Y 63.3649, Z -5.5000, A 0.000, B 0.000, C 0.000 }
gfCNCPoint4[1987] = {X 549.9934, Y 62.1585, Z -5.5000, A 0.000, B 0.000, C 0.000 }
gfCNCPoint4[1988] = {X 548.2696, Y 60.7644, Z -5.5000, A 0.000, B 0.000, C 0.000 }
gfCNCPoint4[1989] = {X 546.7008, Y 59.1979, Z -5.5000, A 0.000, B 0.000, C 0.000 }
gfCNCPoint4[1990] = {X 545.1842, Y 59.4178, Z -5.5000, A 0.000, B 0.000, C 0.000 }
gfCNCPoint4[1991] = {X 543.6528, Y 59.4763, Z -5.5000, A 0.000, B 0.000, C 0.000 }
gfCNCPoint4[1992] = {X 527.5782, Y 59.4766, Z -5.5000, A 0.000, B 0.000, C 0.000 }
gfCNCPoint4[1993] = {X 525.9242, Y 60.2757, Z -5.5000, A 0.000, B 0.000, C 0.000 }
gfCNCPoint4[1994] = {X 524.1831, Y 60.8614, Z -5.5000, A 0.000, B 0.000, C 0.000 }
gfCNCPoint4[1995] = {X 522.3823, Y 61.2243, Z -5.5000, A 0.000, B 0.000, C 0.000 }
gfCNCPoint4[1996] = {X 520.5503, Y 61.3589, Z -5.5000, A 0.000, B 0.000, C 0.000 }
gfCNCPoint4[1997] = {X 519.7998, Y 61.3591, Z -5.5000, A 0.000, B 0.000, C 0.000 }
gfCNCPoint4[1998] = {X 518.0043, Y 61.2474, Z -5.5000, A 0.000, B 0.000, C 0.000 }
gfCNCPoint4[1999] = {X 516.2365, Y 60.9138, Z -5.5000, A 0.000, B 0.000, C 0.000 }
gfCNCPoint4[2000] = {X 514.5237, Y 60.3637, Z -5.5000, A 0.000, B 0.000, C 0.000 }
gfCNCPoint4[2001] = {X 512.8923, Y 59.6054, Z -5.5000, A 0.000, B 0.000, C 0.000 }
gfCNCPoint4[2002] = {X 511.3676, Y 58.6507, Z -5.5000, A 0.000, B 0.000, C 0.000 }
gfCNCPoint4[2003] = {X 509.9730, Y 57.5142, Z -5.5000, A 0.000, B 0.000, C 0.000 }
gfCNCPoint4[2004] = {X 508.6156, Y 58.2113, Z -5.5000, A 0.000, B 0.000, C 0.000 }
gfCNCPoint4[2005] = {X 507.1924, Y 58.7617, Z -5.5000, A 0.000, B 0.000, C 0.000 }
gfCNCPoint4[2006] = {X 505.7192, Y 59.1593, Z -5.5000, A 0.000, B 0.000, C 0.000 }
gfCNCPoint4[2007] = {X 504.2123, Y 59.3996, Z -5.5000, A 0.000, B 0.000, C 0.000 }
gfCNCPoint4[2008] = {X 502.6885, Y 59.4800, Z -5.5000, A 0.000, B 0.000, C 0.000 }
gfCNCPoint4[2009] = {X 496.2450, Y 59.4800, Z -5.5000, A 0.000, B 0.000, C 0.000 }
gfCNCPoint4[2010] = {X 495.2580, Y 59.4463, Z -5.5000, A 0.000, B 0.000, C 0.000 }
gfCNCPoint4[2011] = {X 494.2756, Y 59.3454, Z -5.5000, A 0.000, B 0.000, C 0.000 }
gfCNCPoint4[2012] = {X 494.1342, Y 61.3005, Z -5.5000, A 0.000, B 0.000, C 0.000 }
gfCNCPoint4[2013] = {X 493.7951, Y 63.2310, Z -5.5000, A 0.000, B 0.000, C 0.000 }
gfCNCPoint4[2014] = {X 493.2616, Y 65.1172, Z -5.5000, A 0.000, B 0.000, C 0.000 }
gfCNCPoint4[2015] = {X 492.5395, Y 66.9394, Z -5.5000, A 0.000, B 0.000, C 0.000 }
gfCNCPoint4[2016] = {X 491.6360, Y 68.6789, Z -5.5000, A 0.000, B 0.000, C 0.000 }
gfCNCPoint4[2017] = {X 490.5606, Y 70.3177, Z -5.5000, A 0.000, B 0.000, C 0.000 }
gfCNCPoint4[2018] = {X 490.5608, Y 83.2951, Z -5.5000, A 0.000, B 0.000, C 0.000 }
gfCNCPoint4[2019] = {X 507.6814, Y 83.2951, Z -5.5000, A 0.000, B 0.000, C 0.000 }
gfCNCPoint4[2020] = {X 507.6814, Y 85.6951, Z -5.5000, A 0.000, B 0.000, C 0.000 }
gfCNCPoint4[2021] = {X 585.6966, Y 85.6951, Z -5.5000, A 0.000, B 0.000, C 0.000 }
gfCNCPoint4[2022] = {X 585.6966, Y 63.3150, Z -5.5000, A 0.000, B 0.000, C 0.000 }
gfCNCPoint4[2023] = {X 584.3996, Y 63.5678, Z -5.5000, A 0.000, B 0.000, C 0.000 }
gfCNCPoint4[2024] = {X 583.0880, Y 63.7288, Z -5.5000, A 0.000, B 0.000, C 0.000 }
gfCNCPoint4[2025] = {X 581.1243, Y 63.7971, Z -5.5000, A 0.000, B 0.000, C 0.000 }
gfCNCPoint4[2026] = {X 579.1642, Y 63.6600, Z -5.5000, A 0.000, B 0.000, C 0.000 }
gfCNCPoint4[2027] = {X 577.2291, Y 63.3191, Z -5.5000, A 0.000, B 0.000, C 0.000 }
gfCNCPoint4[2028] = {X 575.3401, Y 62.7781, Z -5.5000, A 0.000, B 0.000, C 0.000 }
gfCNCPoint4[2029] = {X 573.3441, Y 63.3435, Z -5.5000, A 0.000, B 0.000, C 0.000 }
gfCNCPoint4[2030] = {X 571.2979, Y 63.6855, Z -5.5000, A 0.000, B 0.000, C 0.000 }
gfCNCPoint4[2031] = {X 569.2264, Y 63.8000, Z -5.5000, A 0.000, B 0.000, C 0.000 }
gfCNCPoint4[2032] = {X 562.4443, Y 63.8000, Z -5.5000, A 0.000, B 0.000, C 0.000 }
gfCNCPoint4[2033] = {X 560.5408, Y 63.7034, Z -5.5000, A 0.000, B 0.000, C 0.000 }
gfCNCPoint4[2034] = {X 558.6569, Y 63.4145, Z -5.5000, A 0.000, B 0.000, C 0.000 }
gfCNCPoint4[2035] = {X 556.8119, Y 62.9364, Z -5.5000, A 0.000, B 0.000, C 0.000 }
gfCNCPoint4[2036] = {X 555.0248, Y 62.2740, Z -5.5000, A 0.000, B 0.000, C 0.000 }
gfCNCPoint4[2037] = {X 553.3140, Y 61.4340, Z -5.5000, A 0.000, B 0.000, C 0.000 }
gfCNCPoint4[2038] = {X 551.6970, Y 60.4251, Z -5.5000, A 0.000, B 0.000, C 0.000 }
gfCNCPoint4[2039] = {X 550.1904, Y 59.2577, Z -5.5000, A 0.000, B 0.000, C 0.000 }
gfCNCPoint4[2040] = {X 548.8098, Y 57.9437, Z -5.5000, A 0.000, B 0.000, C 0.000 }
gfCNCPoint4[2041] = {X 547.5693, Y 56.4967, Z -5.5000, A 0.000, B 0.000, C 0.000 }
gfCNCPoint4[2042] = {X 546.2937, Y 56.8317, Z -5.5000, A 0.000, B 0.000, C 0.000 }
gfCNCPoint4[2043] = {X 544.9892, Y 57.0256, Z -5.5000, A 0.000, B 0.000, C 0.000 }
gfCNCPoint4[2044] = {X 543.6713, Y 57.0763, Z -5.5000, A 0.000, B 0.000, C 0.000 }
gfCNCPoint4[2045] = {X 526.9186, Y 57.0766, Z -5.5000, A 0.000, B 0.000, C 0.000 }
gfCNCPoint4[2046] = {X 525.4333, Y 57.8749, Z -5.5000, A 0.000, B 0.000, C 0.000 }
gfCNCPoint4[2047] = {X 523.8524, Y 58.4615, Z -5.5000, A 0.000, B 0.000, C 0.000 }
gfCNCPoint4[2048] = {X 522.2058, Y 58.8251, Z -5.5000, A 0.000, B 0.000, C 0.000 }
gfCNCPoint4[2049] = {X 520.5249, Y 58.9590, Z -5.5000, A 0.000, B 0.000, C 0.000 }
gfCNCPoint4[2050] = {X 519.7998, Y 58.9591, Z -5.5000, A 0.000, B 0.000, C 0.000 }
gfCNCPoint4[2051] = {X 518.2467, Y 58.8589, Z -5.5000, A 0.000, B 0.000, C 0.000 }
gfCNCPoint4[2052] = {X 516.7195, Y 58.5598, Z -5.5000, A 0.000, B 0.000, C 0.000 }
gfCNCPoint4[2053] = {X 515.2433, Y 58.0668, Z -5.5000, A 0.000, B 0.000, C 0.000 }
gfCNCPoint4[2054] = {X 513.8428, Y 57.3882, Z -5.5000, A 0.000, B 0.000, C 0.000 }
gfCNCPoint4[2055] = {X 512.5411, Y 56.5351, Z -5.5000, A 0.000, B 0.000, C 0.000 }
gfCNCPoint4[2056] = {X 511.3600, Y 55.5218, Z -5.5000, A 0.000, B 0.000, C 0.000 }
gfCNCPoint4[2057] = {X 510.3189, Y 54.3650, Z -5.5000, A 0.000, B 0.000, C 0.000 }
gfCNCPoint4[2058] = {X 508.9711, Y 55.3177, Z -5.5000, A 0.000, B 0.000, C 0.000 }
gfCNCPoint4[2059] = {X 507.5060, Y 56.0778, Z -5.5000, A 0.000, B 0.000, C 0.000 }
gfCNCPoint4[2060] = {X 505.9510, Y 56.6311, Z -5.5000, A 0.000, B 0.000, C 0.000 }
gfCNCPoint4[2061] = {X 504.3351, Y 56.9672, Z -5.5000, A 0.000, B 0.000, C 0.000 }
gfCNCPoint4[2062] = {X 502.6885, Y 57.0800, Z -5.5000, A 0.000, B 0.000, C 0.000 }
gfCNCPoint4[2063] = {X 496.2450, Y 57.0800, Z -5.5000, A 0.000, B 0.000, C 0.000 }
gfCNCPoint4[2064] = {X 495.4216, Y 57.0519, Z -5.5000, A 0.000, B 0.000, C 0.000 }
gfCNCPoint4[2065] = {X 494.6020, Y 56.9677, Z -5.5000, A 0.000, B 0.000, C 0.000 }
gfCNCPoint4[2066] = {X 493.1719, Y 56.6826, Z -5.5000, A 0.000, B 0.000, C 0.000 }
gfCNCPoint4[2067] = {X 491.7866, Y 56.2272, Z -5.5000, A 0.000, B 0.000, C 0.000 }
gfCNCPoint4[2068] = {X 491.8566, Y 57.1124, Z -5.5000, A 0.000, B 0.000, C 0.000 }
gfCNCPoint4[2069] = {X 491.8800, Y 58.0000, Z -5.5000, A 0.000, B 0.000, C 0.000 }
gfCNCPoint4[2070] = {X 491.8794, Y 59.0735, Z -5.5000, A 0.000, B 0.000, C 0.000 }
gfCNCPoint4[2071] = {X 491.8781, Y 59.1839, Z -5.5000, A 0.000, B 0.000, C 0.000 }
gfCNCPoint4[2072] = {X 491.8762, Y 59.2942, Z -5.5000, A 0.000, B 0.000, C 0.000 }
gfCNCPoint4[2073] = {X 491.7363, Y 61.1317, Z -5.5000, A 0.000, B 0.000, C 0.000 }
gfCNCPoint4[2074] = {X 491.3970, Y 62.9430, Z -5.5000, A 0.000, B 0.000, C 0.000 }
gfCNCPoint4[2075] = {X 490.8623, Y 64.7065, Z -5.5000, A 0.000, B 0.000, C 0.000 }
gfCNCPoint4[2076] = {X 490.1386, Y 66.4012, Z -5.5000, A 0.000, B 0.000, C 0.000 }
gfCNCPoint4[2077] = {X 489.2344, Y 68.0069, Z -5.5000, A 0.000, B 0.000, C 0.000 }
gfCNCPoint4[2078] = {X 488.1606, Y 69.5045, Z -5.5000, A 0.000, B 0.000, C 0.000 }
gfCNCPoint4[2079] = {X 488.1608, Y 85.6951, Z -5.5000, A 0.000, B 0.000, C 0.000 }
gfCNCPoint4[2080] = {X 507.6814, Y 85.6951, Z -5.5000, A 0.000, B 0.000, C 0.000 }
gfCNCPoint4[2081] = {X 507.6814, Y 88.0951, Z -5.5000, A 0.000, B 0.000, C 0.000 }
gfCNCPoint4[2082] = {X 588.0966, Y 88.0951, Z -5.5000, A 0.000, B 0.000, C 0.000 }
gfCNCPoint4[2083] = {X 588.0966, Y 60.4644, Z -5.5000, A 0.000, B 0.000, C 0.000 }
gfCNCPoint4[2084] = {X 587.7998, Y 60.3564, Z -5.5000, A 0.000, B 0.000, C 0.000 }
gfCNCPoint4[2085] = {X 587.5052, Y 60.2427, Z -5.5000, A 0.000, B 0.000, C 0.000 }
gfCNCPoint4[2086] = {X 586.3439, Y 60.6540, Z -5.5000, A 0.000, B 0.000, C 0.000 }
gfCNCPoint4[2087] = {X 585.1550, Y 60.9769, Z -5.5000, A 0.000, B 0.000, C 0.000 }
gfCNCPoint4[2088] = {X 583.5153, Y 61.2699, Z -5.5000, A 0.000, B 0.000, C 0.000 }
gfCNCPoint4[2089] = {X 581.8543, Y 61.3951, Z -5.5000, A 0.000, B 0.000, C 0.000 }
gfCNCPoint4[2090] = {X 580.1893, Y 61.3512, Z -5.5000, A 0.000, B 0.000, C 0.000 }
gfCNCPoint4[2091] = {X 578.5372, Y 61.1386, Z -5.5000, A 0.000, B 0.000, C 0.000 }
gfCNCPoint4[2092] = {X 576.9153, Y 60.7595, Z -5.5000, A 0.000, B 0.000, C 0.000 }
gfCNCPoint4[2093] = {X 575.3401, Y 60.2178, Z -5.5000, A 0.000, B 0.000, C 0.000 }
gfCNCPoint4[2094] = {X 573.8611, Y 60.7315, Z -5.5000, A 0.000, B 0.000, C 0.000 }
gfCNCPoint4[2095] = {X 572.3399, Y 61.1017, Z -5.5000, A 0.000, B 0.000, C 0.000 }
gfCNCPoint4[2096] = {X 570.7903, Y 61.3253, Z -5.5000, A 0.000, B 0.000, C 0.000 }
gfCNCPoint4[2097] = {X 569.2264, Y 61.4000, Z -5.5000, A 0.000, B 0.000, C 0.000 }
gfCNCPoint4[2098] = {X 562.4443, Y 61.4000, Z -5.5000, A 0.000, B 0.000, C 0.000 }
gfCNCPoint4[2099] = {X 560.5829, Y 61.2940, Z -5.5000, A 0.000, B 0.000, C 0.000 }
gfCNCPoint4[2100] = {X 558.7455, Y 60.9775, Z -5.5000, A 0.000, B 0.000, C 0.000 }
gfCNCPoint4[2101] = {X 556.9560, Y 60.4544, Z -5.5000, A 0.000, B 0.000, C 0.000 }
gfCNCPoint4[2102] = {X 555.2374, Y 59.7316, Z -5.5000, A 0.000, B 0.000, C 0.000 }
gfCNCPoint4[2103] = {X 553.6119, Y 58.8184, Z -5.5000, A 0.000, B 0.000, C 0.000 }
gfCNCPoint4[2104] = {X 552.1006, Y 57.7266, Z -5.5000, A 0.000, B 0.000, C 0.000 }
gfCNCPoint4[2105] = {X 550.7229, Y 56.4704, Z -5.5000, A 0.000, B 0.000, C 0.000 }
gfCNCPoint4[2106] = {X 549.4968, Y 55.0659, Z -5.5000, A 0.000, B 0.000, C 0.000 }
gfCNCPoint4[2107] = {X 548.4380, Y 53.5313, Z -5.5000, A 0.000, B 0.000, C 0.000 }
gfCNCPoint4[2108] = {X 547.3161, Y 54.0429, Z -5.5000, A 0.000, B 0.000, C 0.000 }
gfCNCPoint4[2109] = {X 546.1382, Y 54.4078, Z -5.5000, A 0.000, B 0.000, C 0.000 }
gfCNCPoint4[2110] = {X 544.9236, Y 54.6200, Z -5.5000, A 0.000, B 0.000, C 0.000 }
gfCNCPoint4[2111] = {X 543.6918, Y 54.6763, Z -5.5000, A 0.000, B 0.000, C 0.000 }
gfCNCPoint4[2112] = {X 526.1844, Y 54.6766, Z -5.5000, A 0.000, B 0.000, C 0.000 }
gfCNCPoint4[2113] = {X 524.8902, Y 55.4732, Z -5.5000, A 0.000, B 0.000, C 0.000 }
gfCNCPoint4[2114] = {X 523.4887, Y 56.0610, Z -5.5000, A 0.000, B 0.000, C 0.000 }
gfCNCPoint4[2115] = {X 522.0134, Y 56.4258, Z -5.5000, A 0.000, B 0.000, C 0.000 }
gfCNCPoint4[2116] = {X 520.4995, Y 56.5591, Z -5.5000, A 0.000, B 0.000, C 0.000 }
gfCNCPoint4[2117] = {X 519.7998, Y 56.5591, Z -5.5000, A 0.000, B 0.000, C 0.000 }
gfCNCPoint4[2118] = {X 518.3493, Y 56.4498, Z -5.5000, A 0.000, B 0.000, C 0.000 }
gfCNCPoint4[2119] = {X 516.9316, Y 56.1244, Z -5.5000, A 0.000, B 0.000, C 0.000 }
gfCNCPoint4[2120] = {X 515.5787, Y 55.5903, Z -5.5000, A 0.000, B 0.000, C 0.000 }
gfCNCPoint4[2121] = {X 514.3210, Y 54.8595, Z -5.5000, A 0.000, B 0.000, C 0.000 }
gfCNCPoint4[2122] = {X 513.1871, Y 53.9484, Z -5.5000, A 0.000, B 0.000, C 0.000 }
gfCNCPoint4[2123] = {X 512.2025, Y 52.8778, Z -5.5000, A 0.000, B 0.000, C 0.000 }
gfCNCPoint4[2124] = {X 511.3855, Y 51.6648, Z -5.5000, A 0.000, B 0.000, C 0.000 }
gfCNCPoint4[2125] = {X 510.7606, Y 50.3426, Z -5.5000, A 0.000, B 0.000, C 0.000 }
gfCNCPoint4[2126] = {X 509.8636, Y 51.4977, Z -5.5000, A 0.000, B 0.000, C 0.000 }
gfCNCPoint4[2127] = {X 508.8029, Y 52.5044, Z -5.5000, A 0.000, B 0.000, C 0.000 }
gfCNCPoint4[2128] = {X 507.7229, Y 53.2678, Z -5.5000, A 0.000, B 0.000, C 0.000 }
gfCNCPoint4[2129] = {X 506.5489, Y 53.8769, Z -5.5000, A 0.000, B 0.000, C 0.000 }
gfCNCPoint4[2130] = {X 505.3028, Y 54.3203, Z -5.5000, A 0.000, B 0.000, C 0.000 }
gfCNCPoint4[2131] = {X 504.0080, Y 54.5896, Z -5.5000, A 0.000, B 0.000, C 0.000 }
gfCNCPoint4[2132] = {X 502.6885, Y 54.6800, Z -5.5000, A 0.000, B 0.000, C 0.000 }
gfCNCPoint4[2133] = {X 496.2450, Y 54.6800, Z -5.5000, A 0.000, B 0.000, C 0.000 }
gfCNCPoint4[2134] = {X 495.0285, Y 54.6033, Z -5.5000, A 0.000, B 0.000, C 0.000 }
gfCNCPoint4[2135] = {X 493.8313, Y 54.3742, Z -5.5000, A 0.000, B 0.000, C 0.000 }
gfCNCPoint4[2136] = {X 492.6724, Y 53.9966, Z -5.5000, A 0.000, B 0.000, C 0.000 }
gfCNCPoint4[2137] = {X 491.4451, Y 53.4062, Z -5.5000, A 0.000, B 0.000, C 0.000 }
gfCNCPoint4[2138] = {X 490.3129, Y 52.6493, Z -5.5000, A 0.000, B 0.000, C 0.000 }
gfCNCPoint4[2139] = {X 489.2980, Y 51.7410, Z -5.5000, A 0.000, B 0.000, C 0.000 }
gfCNCPoint4[2140] = {X 488.8683, Y 52.1573, Z -5.5000, A 0.000, B 0.000, C 0.000 }
gfCNCPoint4[2141] = {X 488.4137, Y 52.5463, Z -5.5000, A 0.000, B 0.000, C 0.000 }
gfCNCPoint4[2142] = {X 488.8649, Y 53.8245, Z -5.5000, A 0.000, B 0.000, C 0.000 }
gfCNCPoint4[2143] = {X 489.1946, Y 55.1393, Z -5.5000, A 0.000, B 0.000, C 0.000 }
gfCNCPoint4[2144] = {X 489.3999, Y 56.4792, Z -5.5000, A 0.000, B 0.000, C 0.000 }
gfCNCPoint4[2145] = {X 489.4600, Y 57.2386, Z -5.5000, A 0.000, B 0.000, C 0.000 }
gfCNCPoint4[2146] = {X 489.4800, Y 58.0000, Z -5.5000, A 0.000, B 0.000, C 0.000 }
gfCNCPoint4[2147] = {X 489.4795, Y 59.0537, Z -5.5000, A 0.000, B 0.000, C 0.000 }
gfCNCPoint4[2148] = {X 489.3596, Y 60.7977, Z -5.5000, A 0.000, B 0.000, C 0.000 }
gfCNCPoint4[2149] = {X 489.0304, Y 62.5145, Z -5.5000, A 0.000, B 0.000, C 0.000 }
gfCNCPoint4[2150] = {X 488.4966, Y 64.1792, Z -5.5000, A 0.000, B 0.000, C 0.000 }
gfCNCPoint4[2151] = {X 487.7662, Y 65.7674, Z -5.5000, A 0.000, B 0.000, C 0.000 }
gfCNCPoint4[2152] = {X 486.8497, Y 67.2560, Z -5.5000, A 0.000, B 0.000, C 0.000 }
gfCNCPoint4[2153] = {X 485.7606, Y 68.6233, Z -5.5000, A 0.000, B 0.000, C 0.000 }
gfCNCPoint4[2154] = {X 485.7608, Y 87.3792, Z -5.5000, A 0.000, B 0.000, C 0.000 }
gfCNCPoint4[2155] = {X 486.0689, Y 87.7322, Z -5.5000, A 0.000, B 0.000, C 0.000 }
gfCNCPoint4[2156] = {X 486.3654, Y 88.0951, Z -5.5000, A 0.000, B 0.000, C 0.000 }
gfCNCPoint4[2157] = {X 507.6814, Y 88.0951, Z -5.5000, A 0.000, B 0.000, C 0.000 }
gfCNCPoint4[2158] = {X 507.6814, Y 90.4951, Z -5.5000, A 0.000, B 0.000, C 0.000 }
gfCNCPoint4[2159] = {X 590.4966, Y 90.4951, Z -5.5000, A 0.000, B 0.000, C 0.000 }
gfCNCPoint4[2160] = {X 590.4966, Y 58.6615, Z -5.5000, A 0.000, B 0.000, C 0.000 }
gfCNCPoint4[2161] = {X 588.9715, Y 58.2279, Z -5.5000, A 0.000, B 0.000, C 0.000 }
gfCNCPoint4[2162] = {X 587.5052, Y 57.6246, Z -5.5000, A 0.000, B 0.000, C 0.000 }
gfCNCPoint4[2163] = {X 585.8387, Y 58.2956, Z -5.5000, A 0.000, B 0.000, C 0.000 }
gfCNCPoint4[2164] = {X 584.0999, Y 58.7477, Z -5.5000, A 0.000, B 0.000, C 0.000 }
gfCNCPoint4[2165] = {X 582.3176, Y 58.9733, Z -5.5000, A 0.000, B 0.000, C 0.000 }
gfCNCPoint4[2166] = {X 580.5210, Y 58.9689, Z -5.5000, A 0.000, B 0.000, C 0.000 }
gfCNCPoint4[2167] = {X 578.7398, Y 58.7344, Z -5.5000, A 0.000, B 0.000, C 0.000 }
gfCNCPoint4[2168] = {X 577.0034, Y 58.2738, Z -5.5000, A 0.000, B 0.000, C 0.000 }
gfCNCPoint4[2169] = {X 575.3401, Y 57.5945, Z -5.5000, A 0.000, B 0.000, C 0.000 }
gfCNCPoint4[2170] = {X 573.8813, Y 58.2035, Z -5.5000, A 0.000, B 0.000, C 0.000 }
gfCNCPoint4[2171] = {X 572.3630, Y 58.6441, Z -5.5000, A 0.000, B 0.000, C 0.000 }
gfCNCPoint4[2172] = {X 570.8048, Y 58.9107, Z -5.5000, A 0.000, B 0.000, C 0.000 }
gfCNCPoint4[2173] = {X 569.2264, Y 59.0000, Z -5.5000, A 0.000, B 0.000, C 0.000 }
gfCNCPoint4[2174] = {X 562.4443, Y 59.0000, Z -5.5000, A 0.000, B 0.000, C 0.000 }
gfCNCPoint4[2175] = {X 560.6577, Y 58.8855, Z -5.5000, A 0.000, B 0.000, C 0.000 }
gfCNCPoint4[2176] = {X 558.9003, Y 58.5440, Z -5.5000, A 0.000, B 0.000, C 0.000 }
gfCNCPoint4[2177] = {X 557.2009, Y 57.9810, Z -5.5000, A 0.000, B 0.000, C 0.000 }
gfCNCPoint4[2178] = {X 555.5872, Y 57.2057, Z -5.5000, A 0.000, B 0.000, C 0.000 }
gfCNCPoint4[2179] = {X 554.0856, Y 56.2308, Z -5.5000, A 0.000, B 0.000, C 0.000 }
gfCNCPoint4[2180] = {X 552.7207, Y 55.0723, Z -5.5000, A 0.000, B 0.000, C 0.000 }
gfCNCPoint4[2181] = {X 551.5148, Y 53.7491, Z -5.5000, A 0.000, B 0.000, C 0.000 }
gfCNCPoint4[2182] = {X 550.4877, Y 52.2828, Z -5.5000, A 0.000, B 0.000, C 0.000 }
gfCNCPoint4[2183] = {X 549.8379, Y 51.0891, Z -5.5000, A 0.000, B 0.000, C 0.000 }
gfCNCPoint4[2184] = {X 549.3069, Y 49.8381, Z -5.5000, A 0.000, B 0.000, C 0.000 }
gfCNCPoint4[2185] = {X 548.3755, Y 50.7150, Z -5.5000, A 0.000, B 0.000, C 0.000 }
gfCNCPoint4[2186] = {X 547.3052, Y 51.4154, Z -5.5000, A 0.000, B 0.000, C 0.000 }
gfCNCPoint4[2187] = {X 546.1636, Y 51.9064, Z -5.5000, A 0.000, B 0.000, C 0.000 }
gfCNCPoint4[2188] = {X 544.9552, Y 52.1961, Z -5.5000, A 0.000, B 0.000, C 0.000 }
gfCNCPoint4[2189] = {X 543.7151, Y 52.2763, Z -5.5000, A 0.000, B 0.000, C 0.000 }
gfCNCPoint4[2190] = {X 525.3423, Y 52.2766, Z -5.5000, A 0.000, B 0.000, C 0.000 }
gfCNCPoint4[2191] = {X 524.2750, Y 53.0681, Z -5.5000, A 0.000, B 0.000, C 0.000 }
gfCNCPoint4[2192] = {X 523.0840, Y 53.6571, Z -5.5000, A 0.000, B 0.000, C 0.000 }
gfCNCPoint4[2193] = {X 521.8071, Y 54.0246, Z -5.5000, A 0.000, B 0.000, C 0.000 }
gfCNCPoint4[2194] = {X 520.4852, Y 54.1591, Z -5.5000, A 0.000, B 0.000, C 0.000 }
gfCNCPoint4[2195] = {X 519.7998, Y 54.1591, Z -5.5000, A 0.000, B 0.000, C 0.000 }
gfCNCPoint4[2196] = {X 518.5529, Y 54.0515, Z -5.5000, A 0.000, B 0.000, C 0.000 }
gfCNCPoint4[2197] = {X 517.3428, Y 53.7320, Z -5.5000, A 0.000, B 0.000, C 0.000 }
gfCNCPoint4[2198] = {X 516.2054, Y 53.2099, Z -5.5000, A 0.000, B 0.000, C 0.000 }
gfCNCPoint4[2199] = {X 515.1742, Y 52.5007, Z -5.5000, A 0.000, B 0.000, C 0.000 }
gfCNCPoint4[2200] = {X 514.2797, Y 51.6254, Z -5.5000, A 0.000, B 0.000, C 0.000 }
gfCNCPoint4[2201] = {X 513.5483, Y 50.6098, Z -5.5000, A 0.000, B 0.000, C 0.000 }
gfCNCPoint4[2202] = {X 513.0017, Y 49.4839, Z -5.5000, A 0.000, B 0.000, C 0.000 }
gfCNCPoint4[2203] = {X 512.7353, Y 48.6374, Z -5.5000, A 0.000, B 0.000, C 0.000 }
gfCNCPoint4[2204] = {X 512.5739, Y 47.7649, Z -5.5000, A 0.000, B 0.000, C 0.000 }
gfCNCPoint4[2205] = {X 512.5198, Y 46.8791, Z -5.5000, A 0.000, B 0.000, C 0.000 }
gfCNCPoint4[2206] = {X 512.5198, Y 39.9011, Z -5.5000, A 0.000, B 0.000, C 0.000 }
gfCNCPoint4[2207] = {X 512.5808, Y 38.9608, Z -5.5000, A 0.000, B 0.000, C 0.000 }
gfCNCPoint4[2208] = {X 512.7627, Y 38.0362, Z -5.5000, A 0.000, B 0.000, C 0.000 }
gfCNCPoint4[2209] = {X 513.0625, Y 37.1429, Z -5.5000, A 0.000, B 0.000, C 0.000 }
gfCNCPoint4[2210] = {X 513.5581, Y 36.1540, Z -5.5000, A 0.000, B 0.000, C 0.000 }
gfCNCPoint4[2211] = {X 514.1978, Y 35.2517, Z -5.5000, A 0.000, B 0.000, C 0.000 }
gfCNCPoint4[2212] = {X 514.9668, Y 34.4567, Z -5.5000, A 0.000, B 0.000, C 0.000 }
gfCNCPoint4[2213] = {X 515.8474, Y 33.7874, Z -5.5000, A 0.000, B 0.000, C 0.000 }
gfCNCPoint4[2214] = {X 513.2415, Y 29.7564, Z -5.5000, A 0.000, B 0.000, C 0.000 }
gfCNCPoint4[2215] = {X 513.5218, Y 29.5806, Z -5.5000, A 0.000, B 0.000, C 0.000 }
gfCNCPoint4[2216] = {X 513.8068, Y 29.4125, Z -5.5000, A 0.000, B 0.000, C 0.000 }
gfCNCPoint4[2217] = {X 513.8068, Y 27.6757, Z -5.5000, A 0.000, B 0.000, C 0.000 }
gfCNCPoint4[2218] = {X 513.5216, Y 27.5012, Z -5.5000, A 0.000, B 0.000, C 0.000 }
gfCNCPoint4[2219] = {X 513.2415, Y 27.3189, Z -5.5000, A 0.000, B 0.000, C 0.000 }
gfCNCPoint4[2220] = {X 513.2415, Y 29.7564, Z -5.5000, A 0.000, B 0.000, C 0.000 }
gfCNCPoint4[2221] = {X 514.5444, Y 31.7719, Z -5.5000, A 0.000, B 0.000, C 0.000 }
gfCNCPoint4[2222] = {X 515.3548, Y 31.3020, Z -5.5000, A 0.000, B 0.000, C 0.000 }
gfCNCPoint4[2223] = {X 516.2068, Y 30.9126, Z -5.5000, A 0.000, B 0.000, C 0.000 }
gfCNCPoint4[2224] = {X 516.2068, Y 26.2046, Z -5.5000, A 0.000, B 0.000, C 0.000 }
gfCNCPoint4[2225] = {X 515.3714, Y 25.8041, Z -5.5000, A 0.000, B 0.000, C 0.000 }
gfCNCPoint4[2226] = {X 514.5781, Y 25.3256, Z -5.5000, A 0.000, B 0.000, C 0.000 }
gfCNCPoint4[2227] = {X 513.5949, Y 24.5708, Z -5.5000, A 0.000, B 0.000, C 0.000 }
gfCNCPoint4[2228] = {X 512.7163, Y 23.6966, Z -5.5000, A 0.000, B 0.000, C 0.000 }
gfCNCPoint4[2229] = {X 511.9565, Y 22.7172, Z -5.5000, A 0.000, B 0.000, C 0.000 }
gfCNCPoint4[2230] = {X 511.3282, Y 21.6488, Z -5.5000, A 0.000, B 0.000, C 0.000 }
gfCNCPoint4[2231] = {X 510.8415, Y 20.5089, Z -5.5000, A 0.000, B 0.000, C 0.000 }
gfCNCPoint4[2232] = {X 510.8415, Y 36.2336, Z -5.5000, A 0.000, B 0.000, C 0.000 }
gfCNCPoint4[2233] = {X 511.5005, Y 34.9188, Z -5.5000, A 0.000, B 0.000, C 0.000 }
gfCNCPoint4[2234] = {X 512.3510, Y 33.7190, Z -5.5000, A 0.000, B 0.000, C 0.000 }
gfCNCPoint4[2235] = {X 513.3736, Y 32.6619, Z -5.5000, A 0.000, B 0.000, C 0.000 }
gfCNCPoint4[2236] = {X 514.5444, Y 31.7719, Z -5.5000, A 0.000, B 0.000, C 0.000 }
gfCNCPoint4[2237] = {X 515.8474, Y 33.7874, Z -5.5000, A 0.000, B 0.000, C 0.000 }
gfCNCPoint4[2238] = {X 516.7439, Y 33.2935, Z -5.5000, A 0.000, B 0.000, C 0.000 }
gfCNCPoint4[2239] = {X 517.7007, Y 32.9303, Z -5.5000, A 0.000, B 0.000, C 0.000 }
gfCNCPoint4[2240] = {X 518.6990, Y 32.7048, Z -5.5000, A 0.000, B 0.000, C 0.000 }
gfCNCPoint4[2241] = {X 518.6299, Y 32.1290, Z -5.5000, A 0.000, B 0.000, C 0.000 }
gfCNCPoint4[2242] = {X 518.6068, Y 31.5495, Z -5.5000, A 0.000, B 0.000, C 0.000 }
gfCNCPoint4[2243] = {X 518.6068, Y 24.5714, Z -5.5000, A 0.000, B 0.000, C 0.000 }
gfCNCPoint4[2244] = {X 518.6080, Y 24.4373, Z -5.5000, A 0.000, B 0.000, C 0.000 }
gfCNCPoint4[2245] = {X 517.3913, Y 24.0940, Z -5.5000, A 0.000, B 0.000, C 0.000 }
gfCNCPoint4[2246] = {X 516.2523, Y 23.5454, Z -5.5000, A 0.000, B 0.000, C 0.000 }
gfCNCPoint4[2247] = {X 515.2254, Y 22.8080, Z -5.5000, A 0.000, B 0.000, C 0.000 }
gfCNCPoint4[2248] = {X 514.3415, Y 21.9040, Z -5.5000, A 0.000, B 0.000, C 0.000 }
gfCNCPoint4[2249] = {X 513.6274, Y 20.8608, Z -5.5000, A 0.000, B 0.000, C 0.000 }
gfCNCPoint4[2250] = {X 513.1045, Y 19.7098, Z -5.5000, A 0.000, B 0.000, C 0.000 }
gfCNCPoint4[2251] = {X 512.7937, Y 18.5154, Z -5.5000, A 0.000, B 0.000, C 0.000 }
gfCNCPoint4[2252] = {X 512.6891, Y 17.2857, Z -5.5000, A 0.000, B 0.000, C 0.000 }
gfCNCPoint4[2253] = {X 512.6891, Y 10.3077, Z -5.5000, A 0.000, B 0.000, C 0.000 }
gfCNCPoint4[2254] = {X 512.7002, Y 9.9057, Z -5.5000, A 0.000, B 0.000, C 0.000 }
gfCNCPoint4[2255] = {X 512.7335, Y 9.5049, Z -5.5000, A 0.000, B 0.000, C 0.000 }
gfCNCPoint4[2256] = {X 509.4591, Y 9.5049, Z -5.5000, A 0.000, B 0.000, C 0.000 }
gfCNCPoint4[2257] = {X 509.7406, Y 10.3719, Z -5.5000, A 0.000, B 0.000, C 0.000 }
gfCNCPoint4[2258] = {X 509.9113, Y 11.2672, Z -5.5000, A 0.000, B 0.000, C 0.000 }
gfCNCPoint4[2259] = {X 509.9685, Y 12.1769, Z -5.5000, A 0.000, B 0.000, C 0.000 }
gfCNCPoint4[2260] = {X 509.9682, Y 13.0462, Z -5.5000, A 0.000, B 0.000, C 0.000 }
gfCNCPoint4[2261] = {X 509.8612, Y 14.2234, Z -5.5000, A 0.000, B 0.000, C 0.000 }
gfCNCPoint4[2262] = {X 509.5651, Y 15.3678, Z -5.5000, A 0.000, B 0.000, C 0.000 }
gfCNCPoint4[2263] = {X 509.0876, Y 16.4492, Z -5.5000, A 0.000, B 0.000, C 0.000 }
gfCNCPoint4[2264] = {X 508.4415, Y 17.4391, Z -5.5000, A 0.000, B 0.000, C 0.000 }
gfCNCPoint4[2265] = {X 508.4414, Y 39.7476, Z -5.5000, A 0.000, B 0.000, C 0.000 }
gfCNCPoint4[2266] = {X 509.0894, Y 40.7409, Z -5.5000, A 0.000, B 0.000, C 0.000 }
gfCNCPoint4[2267] = {X 509.5675, Y 41.8261, Z -5.5000, A 0.000, B 0.000, C 0.000 }
gfCNCPoint4[2268] = {X 509.8631, Y 42.9746, Z -5.5000, A 0.000, B 0.000, C 0.000 }
gfCNCPoint4[2269] = {X 509.9683, Y 44.1558, Z -5.5000, A 0.000, B 0.000, C 0.000 }
gfCNCPoint4[2270] = {X 509.9685, Y 45.0000, Z -5.5000, A 0.000, B 0.000, C 0.000 }
gfCNCPoint4[2271] = {X 509.8909, Y 46.0603, Z -5.5000, A 0.000, B 0.000, C 0.000 }
gfCNCPoint4[2272] = {X 509.6596, Y 47.0980, Z -5.5000, A 0.000, B 0.000, C 0.000 }
gfCNCPoint4[2273] = {X 509.2797, Y 48.0910, Z -5.5000, A 0.000, B 0.000, C 0.000 }
gfCNCPoint4[2274] = {X 508.7593, Y 49.0180, Z -5.5000, A 0.000, B 0.000, C 0.000 }
gfCNCPoint4[2275] = {X 508.0200, Y 49.9571, Z -5.5000, A 0.000, B 0.000, C 0.000 }
gfCNCPoint4[2276] = {X 507.1371, Y 50.7626, Z -5.5000, A 0.000, B 0.000, C 0.000 }
gfCNCPoint4[2277] = {X 506.1343, Y 51.4129, Z -5.5000, A 0.000, B 0.000, C 0.000 }
gfCNCPoint4[2278] = {X 505.0386, Y 51.8902, Z -5.5000, A 0.000, B 0.000, C 0.000 }
gfCNCPoint4[2279] = {X 503.8796, Y 52.1819, Z -5.5000, A 0.000, B 0.000, C 0.000 }
gfCNCPoint4[2280] = {X 502.6885, Y 52.2800, Z -5.5000, A 0.000, B 0.000, C 0.000 }
gfCNCPoint4[2281] = {X 496.2450, Y 52.2800, Z -5.5000, A 0.000, B 0.000, C 0.000 }
gfCNCPoint4[2282] = {X 495.0845, Y 52.1869, Z -5.5000, A 0.000, B 0.000, C 0.000 }
gfCNCPoint4[2283] = {X 493.9538, Y 51.9100, Z -5.5000, A 0.000, B 0.000, C 0.000 }
gfCNCPoint4[2284] = {X 492.8816, Y 51.4564, Z -5.5000, A 0.000, B 0.000, C 0.000 }
gfCNCPoint4[2285] = {X 491.8954, Y 50.8377, Z -5.5000, A 0.000, B 0.000, C 0.000 }
gfCNCPoint4[2286] = {X 491.0204, Y 50.0697, Z -5.5000, A 0.000, B 0.000, C 0.000 }
gfCNCPoint4[2287] = {X 490.2980, Y 49.1989, Z -5.5000, A 0.000, B 0.000, C 0.000 }
gfCNCPoint4[2288] = {X 489.7192, Y 48.2267, Z -5.5000, A 0.000, B 0.000, C 0.000 }
gfCNCPoint4[2289] = {X 489.2980, Y 47.1766, Z -5.5000, A 0.000, B 0.000, C 0.000 }
gfCNCPoint4[2290] = {X 488.8769, Y 48.2267, Z -5.5000, A 0.000, B 0.000, C 0.000 }
gfCNCPoint4[2291] = {X 488.2981, Y 49.1989, Z -5.5000, A 0.000, B 0.000, C 0.000 }
gfCNCPoint4[2292] = {X 487.5756, Y 50.0697, Z -5.5000, A 0.000, B 0.000, C 0.000 }
gfCNCPoint4[2293] = {X 486.8824, Y 50.6978, Z -5.5000, A 0.000, B 0.000, C 0.000 }
gfCNCPoint4[2294] = {X 486.1145, Y 51.2318, Z -5.5000, A 0.000, B 0.000, C 0.000 }
gfCNCPoint4[2295] = {X 485.2843, Y 51.6629, Z -5.5000, A 0.000, B 0.000, C 0.000 }
gfCNCPoint4[2296] = {X 486.0586, Y 53.1385, Z -5.5000, A 0.000, B 0.000, C 0.000 }
gfCNCPoint4[2297] = {X 486.6224, Y 54.7067, Z -5.5000, A 0.000, B 0.000, C 0.000 }
gfCNCPoint4[2298] = {X 486.9651, Y 56.3375, Z -5.5000, A 0.000, B 0.000, C 0.000 }
gfCNCPoint4[2299] = {X 487.0800, Y 58.0000, Z -5.5000, A 0.000, B 0.000, C 0.000 }
gfCNCPoint4[2300] = {X 487.0796, Y 59.0339, Z -5.5000, A 0.000, B 0.000, C 0.000 }
gfCNCPoint4[2301] = {X 486.9596, Y 60.6351, Z -5.5000, A 0.000, B 0.000, C 0.000 }
gfCNCPoint4[2302] = {X 486.6284, Y 62.2063, Z -5.5000, A 0.000, B 0.000, C 0.000 }
gfCNCPoint4[2303] = {X 486.0916, Y 63.7197, Z -5.5000, A 0.000, B 0.000, C 0.000 }
gfCNCPoint4[2304] = {X 485.3589, Y 65.1485, Z -5.5000, A 0.000, B 0.000, C 0.000 }
gfCNCPoint4[2305] = {X 484.4431, Y 66.4675, Z -5.5000, A 0.000, B 0.000, C 0.000 }
gfCNCPoint4[2306] = {X 483.3605, Y 67.6534, Z -5.5000, A 0.000, B 0.000, C 0.000 }
gfCNCPoint4[2307] = {X 483.3609, Y 88.3502, Z -5.5000, A 0.000, B 0.000, C 0.000 }
gfCNCPoint4[2308] = {X 484.3109, Y 89.3712, Z -5.5000, A 0.000, B 0.000, C 0.000 }
gfCNCPoint4[2309] = {X 485.1367, Y 90.4951, Z -5.5000, A 0.000, B 0.000, C 0.000 }
gfCNCPoint4[2310] = {X 507.6814, Y 90.4951, Z -5.5000, A 0.000, B 0.000, C 0.000 }
gfCNCPoint4[2311] = {X 507.6814, Y 92.8951, Z -5.5000, A 0.000, B 0.000, C 0.000 }
gfCNCPoint4[2312] = {X 592.8966, Y 92.8951, Z -5.5000, A 0.000, B 0.000, C 0.000 }
gfCNCPoint4[2313] = {X 592.8966, Y 56.5812, Z -5.5000, A 0.000, B 0.000, C 0.000 }
gfCNCPoint4[2314] = {X 591.4810, Y 56.4128, Z -5.5000, A 0.000, B 0.000, C 0.000 }
gfCNCPoint4[2315] = {X 590.0968, Y 56.0720, Z -5.5000, A 0.000, B 0.000, C 0.000 }
gfCNCPoint4[2316] = {X 588.7648, Y 55.5641, Z -5.5000, A 0.000, B 0.000, C 0.000 }
gfCNCPoint4[2317] = {X 587.5052, Y 54.8965, Z -5.5000, A 0.000, B 0.000, C 0.000 }
gfCNCPoint4[2318] = {X 586.9690, Y 55.2051, Z -5.5000, A 0.000, B 0.000, C 0.000 }
gfCNCPoint4[2319] = {X 586.4171, Y 55.4846, Z -5.5000, A 0.000, B 0.000, C 0.000 }
gfCNCPoint4[2320] = {X 584.8782, Y 56.0830, Z -5.5000, A 0.000, B 0.000, C 0.000 }
gfCNCPoint4[2321] = {X 583.2699, Y 56.4570, Z -5.5000, A 0.000, B 0.000, C 0.000 }
gfCNCPoint4[2322] = {X 581.6248, Y 56.5987, Z -5.5000, A 0.000, B 0.000, C 0.000 }
gfCNCPoint4[2323] = {X 579.9763, Y 56.5055, Z -5.5000, A 0.000, B 0.000, C 0.000 }
gfCNCPoint4[2324] = {X 578.3577, Y 56.1792, Z -5.5000, A 0.000, B 0.000, C 0.000 }
gfCNCPoint4[2325] = {X 576.8018, Y 55.6263, Z -5.5000, A 0.000, B 0.000, C 0.000 }
gfCNCPoint4[2326] = {X 575.3401, Y 54.8581, Z -5.5000, A 0.000, B 0.000, C 0.000 }
gfCNCPoint4[2327] = {X 573.9176, Y 55.6091, Z -5.5000, A 0.000, B 0.000, C 0.000 }
gfCNCPoint4[2328] = {X 572.4049, Y 56.1560, Z -5.5000, A 0.000, B 0.000, C 0.000 }
gfCNCPoint4[2329] = {X 570.8311, Y 56.4885, Z -5.5000, A 0.000, B 0.000, C 0.000 }
gfCNCPoint4[2330] = {X 569.2264, Y 56.6000, Z -5.5000, A 0.000, B 0.000, C 0.000 }
gfCNCPoint4[2331] = {X 562.4443, Y 56.6000, Z -5.5000, A 0.000, B 0.000, C 0.000 }
gfCNCPoint4[2332] = {X 560.8793, Y 56.4939, Z -5.5000, A 0.000, B 0.000, C 0.000 }
gfCNCPoint4[2333] = {X 559.3429, Y 56.1777, Z -5.5000, A 0.000, B 0.000, C 0.000 }
gfCNCPoint4[2334] = {X 557.8632, Y 55.6571, Z -5.5000, A 0.000, B 0.000, C 0.000 }
gfCNCPoint4[2335] = {X 556.4673, Y 54.9416, Z -5.5000, A 0.000, B 0.000, C 0.000 }
gfCNCPoint4[2336] = {X 555.1807, Y 54.0444, Z -5.5000, A 0.000, B 0.000, C 0.000 }
gfCNCPoint4[2337] = {X 554.0269, Y 52.9817, Z -5.5000, A 0.000, B 0.000, C 0.000 }
gfCNCPoint4[2338] = {X 553.0270, Y 51.7731, Z -5.5000, A 0.000, B 0.000, C 0.000 }
gfCNCPoint4[2339] = {X 552.1993, Y 50.4407, Z -5.5000, A 0.000, B 0.000, C 0.000 }
gfCNCPoint4[2340] = {X 551.5590, Y 49.0087, Z -5.5000, A 0.000, B 0.000, C 0.000 }
gfCNCPoint4[2341] = {X 551.1638, Y 47.7037, Z -5.5000, A 0.000, B 0.000, C 0.000 }
gfCNCPoint4[2342] = {X 550.9244, Y 46.3612, Z -5.5000, A 0.000, B 0.000, C 0.000 }
gfCNCPoint4[2343] = {X 550.8443, Y 45.0000, Z -5.5000, A 0.000, B 0.000, C 0.000 }
gfCNCPoint4[2344] = {X 550.8443, Y 44.0554, Z -5.5000, A 0.000, B 0.000, C 0.000 }
gfCNCPoint4[2345] = {X 550.9568, Y 42.4677, Z -5.5000, A 0.000, B 0.000, C 0.000 }
gfCNCPoint4[2346] = {X 551.2849, Y 40.9102, Z -5.5000, A 0.000, B 0.000, C 0.000 }
gfCNCPoint4[2347] = {X 551.8226, Y 39.4121, Z -5.5000, A 0.000, B 0.000, C 0.000 }
gfCNCPoint4[2348] = {X 549.6245, Y 38.4486, Z -5.5000, A 0.000, B 0.000, C 0.000 }
gfCNCPoint4[2349] = {X 549.7927, Y 38.0795, Z -5.5000, A 0.000, B 0.000, C 0.000 }
gfCNCPoint4[2350] = {X 549.9715, Y 37.7154, Z -5.5000, A 0.000, B 0.000, C 0.000 }
gfCNCPoint4[2351] = {X 549.9715, Y 16.9514, Z -5.5000, A 0.000, B 0.000, C 0.000 }
gfCNCPoint4[2352] = {X 549.8036, Y 17.1980, Z -5.5000, A 0.000, B 0.000, C 0.000 }
gfCNCPoint4[2353] = {X 549.6257, Y 17.4375, Z -5.5000, A 0.000, B 0.000, C 0.000 }
gfCNCPoint4[2354] = {X 549.6245, Y 38.4486, Z -5.5000, A 0.000, B 0.000, C 0.000 }
gfCNCPoint4[2355] = {X 551.8226, Y 39.4121, Z -5.5000, A 0.000, B 0.000, C 0.000 }
gfCNCPoint4[2356] = {X 552.0827, Y 38.8587, Z -5.5000, A 0.000, B 0.000, C 0.000 }
gfCNCPoint4[2357] = {X 552.3715, Y 38.3198, Z -5.5000, A 0.000, B 0.000, C 0.000 }
gfCNCPoint4[2358] = {X 552.3715, Y 11.6872, Z -5.5000, A 0.000, B 0.000, C 0.000 }
gfCNCPoint4[2359] = {X 551.6703, Y 10.2331, Z -5.5000, A 0.000, B 0.000, C 0.000 }
gfCNCPoint4[2360] = {X 551.1778, Y 8.6958, Z -5.5000, A 0.000, B 0.000, C 0.000 }
gfCNCPoint4[2361] = {X 550.9035, Y 7.1049, Z -5.5000, A 0.000, B 0.000, C 0.000 }
gfCNCPoint4[2362] = {X 524.2927, Y 7.1049, Z -5.5000, A 0.000, B 0.000, C 0.000 }
gfCNCPoint4[2363] = {X 524.3784, Y 7.2062, Z -5.5000, A 0.000, B 0.000, C 0.000 }
gfCNCPoint4[2364] = {X 524.4614, Y 7.3098, Z -5.5000, A 0.000, B 0.000, C 0.000 }
gfCNCPoint4[2365] = {X 543.7426, Y 7.3102, Z -5.5000, A 0.000, B 0.000, C 0.000 }
gfCNCPoint4[2366] = {X 544.7120, Y 7.3824, Z -5.5000, A 0.000, B 0.000, C 0.000 }
gfCNCPoint4[2367] = {X 545.6478, Y 7.6450, Z -5.5000, A 0.000, B 0.000, C 0.000 }
gfCNCPoint4[2368] = {X 546.5132, Y 8.0877, Z -5.5000, A 0.000, B 0.000, C 0.000 }
gfCNCPoint4[2369] = {X 547.2737, Y 8.6930, Z -5.5000, A 0.000, B 0.000, C 0.000 }
gfCNCPoint4[2370] = {X 547.8993, Y 9.4369, Z -5.5000, A 0.000, B 0.000, C 0.000 }
gfCNCPoint4[2371] = {X 548.3653, Y 10.2899, Z -5.5000, A 0.000, B 0.000, C 0.000 }
gfCNCPoint4[2372] = {X 548.6531, Y 11.2184, Z -5.5000, A 0.000, B 0.000, C 0.000 }
gfCNCPoint4[2373] = {X 548.7514, Y 12.1854, Z -5.5000, A 0.000, B 0.000, C 0.000 }
gfCNCPoint4[2374] = {X 548.7512, Y 13.0237, Z -5.5000, A 0.000, B 0.000, C 0.000 }
gfCNCPoint4[2375] = {X 548.6554, Y 13.9413, Z -5.5000, A 0.000, B 0.000, C 0.000 }
gfCNCPoint4[2376] = {X 548.3887, Y 14.8244, Z -5.5000, A 0.000, B 0.000, C 0.000 }
gfCNCPoint4[2377] = {X 547.9605, Y 15.6415, Z -5.5000, A 0.000, B 0.000, C 0.000 }
gfCNCPoint4[2378] = {X 547.6191, Y 16.1036, Z -5.5000, A 0.000, B 0.000, C 0.000 }
gfCNCPoint4[2379] = {X 547.2258, Y 16.5224, Z -5.5000, A 0.000, B 0.000, C 0.000 }
gfCNCPoint4[2380] = {X 547.2244, Y 40.6631, Z -5.5000, A 0.000, B 0.000, C 0.000 }
gfCNCPoint4[2381] = {X 547.8656, Y 41.4050, Z -5.5000, A 0.000, B 0.000, C 0.000 }
gfCNCPoint4[2382] = {X 548.3455, Y 42.2601, Z -5.5000, A 0.000, B 0.000, C 0.000 }
gfCNCPoint4[2383] = {X 548.6447, Y 43.1939, Z -5.5000, A 0.000, B 0.000, C 0.000 }
gfCNCPoint4[2384] = {X 548.7513, Y 44.1687, Z -5.5000, A 0.000, B 0.000, C 0.000 }
gfCNCPoint4[2385] = {X 548.7514, Y 45.0006, Z -5.5000, A 0.000, B 0.000, C 0.000 }
gfCNCPoint4[2386] = {X 548.6699, Y 45.8823, Z -5.5000, A 0.000, B 0.000, C 0.000 }
gfCNCPoint4[2387] = {X 548.4305, Y 46.7348, Z -5.5000, A 0.000, B 0.000, C 0.000 }
gfCNCPoint4[2388] = {X 548.0411, Y 47.5301, Z -5.5000, A 0.000, B 0.000, C 0.000 }
gfCNCPoint4[2389] = {X 547.5146, Y 48.2419, Z -5.5000, A 0.000, B 0.000, C 0.000 }
gfCNCPoint4[2390] = {X 546.7290, Y 48.9516, Z -5.5000, A 0.000, B 0.000, C 0.000 }
gfCNCPoint4[2391] = {X 545.8089, Y 49.4753, Z -5.5000, A 0.000, B 0.000, C 0.000 }
gfCNCPoint4[2392] = {X 544.7976, Y 49.7884, Z -5.5000, A 0.000, B 0.000, C 0.000 }
gfCNCPoint4[2393] = {X 543.7426, Y 49.8763, Z -5.5000, A 0.000, B 0.000, C 0.000 }
gfCNCPoint4[2394] = {X 524.3237, Y 49.8767, Z -5.5000, A 0.000, B 0.000, C 0.000 }
gfCNCPoint4[2395] = {X 523.7108, Y 50.5155, Z -5.5000, A 0.000, B 0.000, C 0.000 }
gfCNCPoint4[2396] = {X 522.9956, Y 51.0372, Z -5.5000, A 0.000, B 0.000, C 0.000 }
gfCNCPoint4[2397] = {X 522.2000, Y 51.4256, Z -5.5000, A 0.000, B 0.000, C 0.000 }
gfCNCPoint4[2398] = {X 521.3488, Y 51.6688, Z -5.5000, A 0.000, B 0.000, C 0.000 }
gfCNCPoint4[2399] = {X 520.4681, Y 51.7591, Z -5.5000, A 0.000, B 0.000, C 0.000 }
gfCNCPoint4[2400] = {X 519.7998, Y 51.7591, Z -5.5000, A 0.000, B 0.000, C 0.000 }
gfCNCPoint4[2401] = {X 518.8477, Y 51.6654, Z -5.5000, A 0.000, B 0.000, C 0.000 }
gfCNCPoint4[2402] = {X 517.9323, Y 51.3877, Z -5.5000, A 0.000, B 0.000, C 0.000 }
gfCNCPoint4[2403] = {X 517.0886, Y 50.9367, Z -5.5000, A 0.000, B 0.000, C 0.000 }
gfCNCPoint4[2404] = {X 516.3491, Y 50.3298, Z -5.5000, A 0.000, B 0.000, C 0.000 }
gfCNCPoint4[2405] = {X 515.7422, Y 49.5903, Z -5.5000, A 0.000, B 0.000, C 0.000 }
gfCNCPoint4[2406] = {X 515.2912, Y 48.7466, Z -5.5000, A 0.000, B 0.000, C 0.000 }
gfCNCPoint4[2407] = {X 515.0135, Y 47.8312, Z -5.5000, A 0.000, B 0.000, C 0.000 }
gfCNCPoint4[2408] = {X 514.9198, Y 46.8791, Z -5.5000, A 0.000, B 0.000, C 0.000 }
gfCNCPoint4[2409] = {X 514.9198, Y 39.9011, Z -5.5000, A 0.000, B 0.000, C 0.000 }
gfCNCPoint4[2410] = {X 515.0197, Y 38.9186, Z -5.5000, A 0.000, B 0.000, C 0.000 }
gfCNCPoint4[2411] = {X 515.3154, Y 37.9764, Z -5.5000, A 0.000, B 0.000, C 0.000 }
gfCNCPoint4[2412] = {X 515.7947, Y 37.1129, Z -5.5000, A 0.000, B 0.000, C 0.000 }
gfCNCPoint4[2413] = {X 516.4381, Y 36.3637, Z -5.5000, A 0.000, B 0.000, C 0.000 }
gfCNCPoint4[2414] = {X 517.2191, Y 35.7593, Z -5.5000, A 0.000, B 0.000, C 0.000 }
gfCNCPoint4[2415] = {X 518.1058, Y 35.3245, Z -5.5000, A 0.000, B 0.000, C 0.000 }
gfCNCPoint4[2416] = {X 519.0619, Y 35.0772, Z -5.5000, A 0.000, B 0.000, C 0.000 }
gfCNCPoint4[2417] = {X 519.4084, Y 35.0368, Z -5.5000, A 0.000, B 0.000, C 0.000 }
gfCNCPoint4[2418] = {X 519.7568, Y 35.0213, Z -5.5000, A 0.000, B 0.000, C 0.000 }
gfCNCPoint4[2419] = {X 520.5345, Y 35.0216, Z -5.5000, A 0.000, B 0.000, C 0.000 }
gfCNCPoint4[2420] = {X 521.4084, Y 35.1125, Z -5.5000, A 0.000, B 0.000, C 0.000 }
gfCNCPoint4[2421] = {X 522.2517, Y 35.3587, Z -5.5000, A 0.000, B 0.000, C 0.000 }
gfCNCPoint4[2422] = {X 523.0373, Y 35.7521, Z -5.5000, A 0.000, B 0.000, C 0.000 }
gfCNCPoint4[2423] = {X 523.7396, Y 36.2800, Z -5.5000, A 0.000, B 0.000, C 0.000 }
gfCNCPoint4[2424] = {X 524.3359, Y 36.9253, Z -5.5000, A 0.000, B 0.000, C 0.000 }
gfCNCPoint4[2425] = {X 534.0719, Y 36.9257, Z -5.5000, A 0.000, B 0.000, C 0.000 }
gfCNCPoint4[2426] = {X 534.0719, Y 34.5257, Z -5.5000, A 0.000, B 0.000, C 0.000 }
gfCNCPoint4[2427] = {X 530.3960, Y 34.5254, Z -5.5000, A 0.000, B 0.000, C 0.000 }
gfCNCPoint4[2428] = {X 529.7961, Y 35.1739, Z -5.5000, A 0.000, B 0.000, C 0.000 }
gfCNCPoint4[2429] = {X 529.0891, Y 35.7036, Z -5.5000, A 0.000, B 0.000, C 0.000 }
gfCNCPoint4[2430] = {X 528.2982, Y 36.0972, Z -5.5000, A 0.000, B 0.000, C 0.000 }
gfCNCPoint4[2431] = {X 527.4493, Y 36.3418, Z -5.5000, A 0.000, B 0.000, C 0.000 }
gfCNCPoint4[2432] = {X 526.5703, Y 36.4293, Z -5.5000, A 0.000, B 0.000, C 0.000 }
gfCNCPoint4[2433] = {X 525.8868, Y 36.4294, Z -5.5000, A 0.000, B 0.000, C 0.000 }
